# B&R Automation Studio project PLC code - cp (part 9)

#### LocalFunctions.fun
```iecst
{REDUND_ERROR} FUNCTION ModuleStatus : NIRAdphos_ModuleState (*TODO: Add your comment here*) (*$GROUP=User,$CAT=User,$GROUPICON=User.png,$CATICON=User.png*)
	VAR_INPUT
		StatusValue : INT;
	END_VAR
END_FUNCTION
```

#### Alarms.st
```iecst
ACTION Alarms:

	//////////////////////////
	////// RESET ALARMS //////
	IF data.Commands.xReset THEN
		data.Alarms := resetedAlarms;
		data.AlSummary := resetedAlarmsSummary;
	END_IF

	IF NOT data.Status.xCommsOK THEN
		data.Alarms.xCommsError := TRUE;
	END_IF

	IF data.Signals.In.xFault THEN
		data.Alarms.xFault := TRUE;
	END_IF

	IF NOT data.Signals.In.xSafetyOK THEN
		data.Alarms.xSafetyError := TRUE;
	END_IF

	//Module alarms
	xAnyBlockedFan := FALSE;
	xAnyJam := FALSE;
	FOR iIndexModule := 1 TO data.Parameters.iTotalModules DO

		//Temperatures
		IF data.Status.rSurfaceTempModule[iIndexModule] > data.Parameters.rMaxSurfaceTemp THEN
			data.Alarms.xMaxSurfaceTempModule[iIndexModule] := TRUE;
		END_IF
		IF data.Signals.In.xSurfaceTempModuleSensorError[iIndexModule] THEN
			data.Alarms.xSurfaceTempModuleSensorError[iIndexModule] := TRUE;
		END_IF

		IF data.Signals.In.Jam[iIndexModule].xMechCross AND data.Orders.xCheckJam THEN
			data.Alarms.Jam[iIndexModule].xMechCross:=TRUE;
		END_IF

		//Jams. Check anyJam
		IF data.Alarms.Jam[iIndexModule].xMechCross THEN
			xAnyJam := TRUE;
		END_IF

		//Blocked Fans
		FOR iIndexFan := 1 TO 4 DO
			IF data.Signals.In.BlockedFans[iIndexModule].Fan[iIndexFan] THEN
				data.Alarms.BlockedFansModule[iIndexModule].Fan[iIndexFan] := TRUE;
				xAnyBlockedFan := TRUE;
			END_IF
		END_FOR

	END_FOR

	data.Alarms.xAnyJam := xAnyJam;

	IF data.Signals.In.xInletHumiditySensorError THEN
		data.Alarms.xInletHumiditySensorError := TRUE;
	END_IF
	IF data.Signals.In.xInletTempSensorError THEN
		data.Alarms.xInletTempSensorError := TRUE;
	END_IF

	/////////////////////////////////////////////////////////////////
	//  SOUND  SOUND  SOUND  SOUND  SOUND  SOUND  SOUND
	/////////////////////////////////////////////////////////////////

	arFault(xAlarm:= data.Alarms.xFault, xSilence:=data.Commands.xMute);
	arSafety(xAlarm:= data.Alarms.xSafetyError, xSilence:=data.Commands.xMute);
	arSurfaceTemp1(xAlarm:= data.Alarms.xMaxSurfaceTempModule[1], xSilence:=data.Commands.xMute);
	arSurfaceTemp2(xAlarm:= data.Alarms.xMaxSurfaceTempModule[2], xSilence:=data.Commands.xMute);
	arSurfaceTempSensorError1(xAlarm:= data.Alarms.xSurfaceTempModuleSensorError[1], xSilence:=data.Commands.xMute);
	arSurfaceTempSensorError2(xAlarm:= data.Alarms.xSurfaceTempModuleSensorError[2], xSilence:=data.Commands.xMute);
	arAnyBlockedFan(xAlarm:= xAnyBlockedFan, xSilence:=data.Commands.xMute);
	arAnyJam(xAlarm:= xAnyJam, xSilence:=data.Commands.xMute);

	reasonSound.0 := arFault.xAlarmSound;
	reasonSound.1 := arSafety.xAlarmSound;
	reasonSound.2 := arSurfaceTemp1.xAlarmSound;
	reasonSound.3 := arSurfaceTemp2.xAlarmSound;
	reasonSound.4 := arSurfaceTempSensorError1.xAlarmSound;
	reasonSound.5 := arSurfaceTempSensorError2.xAlarmSound;
	reasonSound.6 := arAnyBlockedFan.xAlarmSound;
	reasonSound.7 := arAnyJam.xAlarmSound;

	data.AlSummary.xAlarmSound := reasonSound>0;

END_ACTION
```

#### AlarmsSummary.st
```iecst
ACTION AlarmsSummary:

	iReasonStop.0 := data.Alarms.xCommsError;
	iReasonStop.1 := data.Alarms.xMaxSurfaceTempModule[1];
	iReasonStop.2 := data.Alarms.xMaxSurfaceTempModule[2];
	iReasonStop.3 := data.Alarms.xFault;
	iReasonStop.4 := data.Alarms.xAnyJam;
	iReasonStop.5 := data.Alarms.xOpcUaWriteError[1] AND data.Status.xEnabledDDC;
	iReasonStop.6 := data.Alarms.xOpcUaWriteError[2] AND data.Status.xEnabledDDC;
	iReasonStop.7 := FALSE;

	data.AlSummary.xAlarmStop := iReasonStop > 0 AND data.Status.xEnabledNir;
	IF EDGEPOS(data.AlSummary.xAlarmStop) THEN
		data.AlSummary.iReasonStop[0] := iReasonStop;
		LogStopAlarm;
	ELSIF EDGEPOS(NOT data.Parameters.AutoMode.xStop AND NOT data.AlSummary.xAlarmStop) THEN
		data.AlSummary.iReasonStop[0] := 0;
	END_IF

	iReasonCritical.0 := data.Status.Comms.Modules[1].error;
	iReasonCritical.1 := data.Status.Comms.Modules[2].error;
	iReasonCritical.2 := data.Alarms.xSafetyError;

	data.AlSummary.xAlarmCritical := iReasonCritical > 0 AND data.Status.xEnabledNir;
	IF EDGEPOS(data.AlSummary.xAlarmCritical) THEN
		data.AlSummary.iReasonCritical := iReasonCritical;
		LogCriticalAlarm;
	ELSIF EDGEPOS(data.Parameters.StateMode=PRINTERGEN_AUTO AND NOT data.AlSummary.xAlarmCritical) THEN
		data.AlSummary.iReasonCritical := 0;
	END_IF

	// It is just used for drive alarms
	iAnyAlarm.0 := iReasonStop > 0;
	iAnyAlarm.1 := iReasonCritical > 0;
	data.AlSummary.xAnyAlarm:= 	iAnyAlarm > 0;

	// It is just used for drive alarms
	iAnyWarning.0 := FALSE;
	data.AlSummary.xAnyWarning:= iAnyWarning > 0;

END_ACTION
```

#### Calculations.st
```iecst
ACTION Calculations:

	//Avoid access out of the array
	data.Parameters.iTotalModules := MIN(data.Parameters.iTotalModules, MAX_LAST_NIR_MODULES);
	data.Parameters.DDC.iLampsExtend := MIN(data.Parameters.DDC.iLampsExtend, 3); //Limit to 3 as make no sense allow higher values

	data.Status.Comms.xBeltRunning := data.Status.Comms.Speed > 1;

	//Calculation of Modules data
	FOR iIndexModule := 1 TO data.Parameters.iTotalModules DO
		data.Status.rSurfaceTempModule[iIndexModule] := INT_TO_REAL(data.Signals.In.iSurfaceTempModuleRaw[iIndexModule])/10.0;
		data.Status.Comms.Modules[iIndexModule].xPowered := data.Status.Comms.Modules[iIndexModule].Power > 1;
		data.Status.Comms.Modules[iIndexModule].NirStatus := ModuleStatus(data.Status.Comms.Modules[iIndexModule].iNirStatus);

		//Limitation of wrong data in parameters
		data.Parameters.Comms.Modules[iIndexModule].Adjust := LIMIT(-100, data.Parameters.Comms.Modules[iIndexModule].Adjust, 100);
	END_FOR;

	data.Status.xDrying := data.State = NIRADPEW_RUNNING;

	// -40C to +60C Probe. 100C Range
	data.Status.rInletTemperature := ((INT_TO_REAL(data.Signals.In.iInletTempRaw)* 100.0)/32767.0)-40.0;
	data.Status.rInletHumidity := ((INT_TO_REAL(data.Signals.In.iInletHumidityRaw)* 100.0)/32767.0)-0.0;

	//Limitations of values to remain consistent
	data.Parameters.Comms.Pstart := MAX(data.Parameters.Comms.Pstart, 0);
	data.Parameters.Comms.Pend := MIN(data.Parameters.Comms.Pend, 100);

	data.Parameters.Comms.Pstart := MIN(data.Parameters.Comms.Pend,data.Parameters.Comms.Pstart);
	data.Parameters.Comms.Pend := MAX(data.Parameters.Comms.Pend,data.Parameters.Comms.Pstart);
	data.Parameters.Comms.Vstart := MIN(data.Parameters.Comms.Vend,data.Parameters.Comms.Vstart);
	data.Parameters.Comms.Vend := MAX(data.Parameters.Comms.Vend,data.Parameters.Comms.Vstart);

	IF data.Parameters.rBeltSpeed > data.Parameters.Comms.Vstart THEN
		data.Status.rPowerSetPoint := data.Parameters.Comms.Pstart +
								(data.Parameters.rBeltSpeed-data.Parameters.Comms.Vstart) *
								(data.Parameters.Comms.Pend-data.Parameters.Comms.Pstart) /
								(data.Parameters.Comms.Vend-data.Parameters.Comms.Vstart);

		IF data.Parameters.xLineEmptyingBelt THEN
			data.Status.rPowerSetPoint := data.Status.rPowerSetPoint * 0.5;
		END_IF
	ELSE
		data.Status.rPowerSetPoint := 0;
	END_IF

END_ACTION
```

#### CommsBase.st
```iecst
ACTION CommsNir1base:

	(* UA_Write - call methode *)
	IndexRange_Nir1.StartIndex := 0;
	IndexRange_Nir1.EndIndex := 47;
	NodeAddInfo_Nir1.AttributeId := UAAI_Value;
	NodeAddInfo_Nir1.IndexRangeCount := 1;
	NodeAddInfo_Nir1.IndexRange[0] := IndexRange_Nir1;
	UA_Write_Nir1(Execute := ExecuteMethodCall_Nir1,
		ConnectionHdl := ConnectionHdl_Nir1,
		NodeHdl := NodeHdl_Nir1,
		NodeAddInfo := NodeAddInfo_Nir1,
		Timeout := T#10s,
		Variable := '::NIRAdphosC.iValues_Nir1'
	);
	IF NOT UA_Write_Nir1.Busy THEN
		ExecuteMethodCall_Nir1 := FALSE;
		IF UA_Write_Nir1.Done THEN
			NewMediaData_Nir1.rLength := NewMediaData_Nir1.rLength + 1;
		END_IF
		IF UA_Write_Nir1.Error THEN
			NewMediaData_Nir1.rDocLength := NewMediaData_Nir1.rDocLength + 1;
		END_IF
	END_IF

//	// Managing the automatic sending. Not sending if enable drying. Sendign Energy then
//	IF NOT gThicknessCtrl.status.xNewMediaStackEnabled OR gThicknessCtrl.parameters.Dry.xDryStack THEN
//		RETURN;
//	END_IF
//
//	IF (gSimMachine.Parameters.Stack.iMediaQuantityToKeepLoaded <= gThicknessCtrl.status.Stack.iNewMediaLoadedL1 + gThicknessCtrl.status.Stack.iNewMediaLoadedL2) THEN
//		RETURN;
//	END_IF

	// Adding a timer to avoid not working the method
//	tonNotCallingMethod_Nir1.IN := NOT UA_Write_Nir1.Busy;
//	tonNotCallingMethod_Nir1.PT := t#4500ms;
//	tonNotCallingMethod_Nir1();
//	IF EDGEPOS(tonNotCallingMethod_Nir1.Q) THEN
//		ExecuteMethodCall_Nir1 := TRUE;
//	END_IF

	IF xReConnect THEN
		PreparingMethodCommsNir1base;
	END_IF

END_ACTION

ACTION InitialDataForMediaNir1base:

END_ACTION

ACTION PreparingMethodCommsNir1base:

	ExecuteConnect_Nir1 := TRUE;

	(* UA_Connect - establish connection to OPC UA Server *)
	SessionConnectInfo_Nir1.SecurityMsgMode := UASecurityMsgMode_None;
	SessionConnectInfo_Nir1.SecurityPolicy := UASecurityPolicy_None;
	SessionConnectInfo_Nir1.TransportProfile := UATP_UATcp;
	SessionConnectInfo_Nir1.UserIdentityToken.UserIdentityTokenType := UAUITT_Anonymous;
	//SessionConnectInfo_Nir1.UserIdentityToken.TokenParam1 := 'PressCore';
	//SessionConnectInfo_Nir1.UserIdentityToken.TokenParam2 := 'h98o76';
	SessionConnectInfo_Nir1.SessionTimeout := T#1m;
	SessionConnectInfo_Nir1.MonitorConnection := T#10s;

	UA_Connect_Nir1(Execute := ExecuteConnect_Nir1,
		ServerEndpointUrl := 'opc.tcp://192.168.125.91:4840',
	SessionConnectInfo := SessionConnectInfo_Nir1,
	Timeout := T#10s);
	IF NOT UA_Connect_Nir1.Busy THEN
		ExecuteConnect_Nir1 := FALSE;
		IF UA_Connect_Nir1.Done THEN
			ConnectionHdl_Nir1 := UA_Connect_Nir1.ConnectionHdl;
			////// NEXT
			ExecuteGetnamespaceindex_Nir1 := TRUE;
		END_IF
		IF UA_Connect_Nir1.Error THEN
			ConnectionHdl_Nir1 := 0;
		END_IF
	END_IF

	(* UA_GetNamespaceIndex - read index of required namespace for PVs *)
	UA_GetNamespaceIndex_Nir1(Execute := ExecuteGetnamespaceindex_Nir1,
		ConnectionHdl := ConnectionHdl_Nir1,
		NamespaceUri := 'http://opcfoundation.org/UA/',
		Timeout := T#5s);
	IF NOT UA_GetNamespaceIndex_Nir1.Busy THEN
		ExecuteGetnamespaceindex_Nir1 := FALSE;
		IF UA_GetNamespaceIndex_Nir1.Done THEN
			NamespaceIndex_Nir1 := UA_GetNamespaceIndex_Nir1.NamespaceIndex;
			////// NEXT
			ExecuteMethodGetHandle_Nir1 := TRUE;
		END_IF
		IF UA_GetNamespaceIndex_Nir1.Error THEN
			NamespaceIndex_Nir1 := 0;
		END_IF
	END_IF

	(* UA_NodeGetHandle - get a handle for required methode *)
	ObjectNodeID_Nir1.NamespaceIndex := NamespaceIndex_Nir1;
	IF NodeHdl_Nir1 = 0 THEN
		ObjectNodeID_Nir1.Identifier := '26';
		ObjectNodeID_Nir1.IdentifierType := UAIdentifierType_Numeric;
	END_IF

	//MethodNodeID_Nir1.NamespaceIndex := NamespaceIndex_Nir1;
	//MethodNodeID_Nir1.Identifier := '::ThickPos:LoadNewMedia';
	//MethodNodeID_Nir1.IdentifierType := UAIdentifierType_String;
	UA_NodeGetHandle_Nir1(Execute := ExecuteMethodGetHandle_Nir1,
		ConnectionHdl := ConnectionHdl_Nir1,
		NodeID := ObjectNodeID_Nir1,
		//MethodNodeID := MethodNodeID_Nir1,
		Timeout := T#10s);
	IF NOT UA_NodeGetHandle_Nir1.Busy THEN
		ExecuteMethodGetHandle_Nir1 := FALSE;
		IF UA_NodeGetHandle_Nir1.Done THEN
			NodeHdl_Nir1 := UA_NodeGetHandle_Nir1.NodeHdl;
			xReConnect := FALSE;
			////// NEXT
			// READY TO COMMUNICATE
		END_IF
		IF UA_NodeGetHandle_Nir1.Error THEN
			NodeHdl_Nir1 := 0;
			xReConnect := FALSE;
		END_IF
	END_IF

	iTimes := iTimes + 1;

END_ACTION
```

#### NIRAdphosCtrl.st
```iecst
PROGRAM _INIT
	data ACCESS ADR(gNirAdphos);
	//Activate this signal because it not exist physically
	data.Signals.In.xSafetyOK := TRUE;

	InitialDataForMediaNir1;
	//PreparingMethodCommsNir1;
	data.Parameters.DDC.pIntensityNir1 := 0;
	data.Parameters.DDC.pIntensityNir2 := 0;

END_PROGRAM

PROGRAM _CYCLIC

	data ACCESS ADR(gNirAdphos);

	Calculations;

	//Consider the parametrization to use NIR or not when ready
	IF (data.State = NIRADPEW_NOT_INITIALIZED OR data.State = NIRADPEW_IDLE) THEN
		data.Status.xEnabledNir := data.Parameters.xEnableNir AND data.Status.xAnyModuleEnabled;
		data.Status.xEnabledDDC := data.Parameters.DDC.xEnableDDC AND data.Status.xAnyModuleEnabled;
	END_IF

	State;

	Alarms;

	AlarmsSummary;

	Outputs;

	CommsNir1;
	CommsNir2;

END_PROGRAM
```

#### NirFunctions.st
```iecst
(* Return Enum from INT value from comms
NIRAdphos_ModuleState
 NIRADPM_OFF				0
 NIRADPM_STARTUP			1
 NIRADPM_READY				2
 NIRADPM_STANDBY			3
 NIRADPM_PROCESS			4
 NIRADPM_SHUTDOWN			5

*)
FUNCTION ModuleStatus
	CASE StatusValue OF
		0: ModuleStatus := NIRADPM_OFF;
		1: ModuleStatus := NIRADPM_STARTUP;
		2: ModuleStatus := NIRADPM_READY;
		3: ModuleStatus := NIRADPM_STANDBY;
		4: ModuleStatus := NIRADPM_PROCESS;
		5: ModuleStatus := NIRADPM_SHUTDOWN;
		ELSE ModuleStatus := NIRADPM_UNDEFINED;
	END_CASE
END_FUNCTION
```

### NirAdphosSim.typ
```iecst
TYPE
	NirAdphosSimParameters_typ : 	STRUCT
		CurrentSpeed : REAL; (*Current speed of the Belt in m/min*)
	END_STRUCT;
	NirAdphosSimCommands_typ : 	STRUCT
		CreateError : BOOL;
	END_STRUCT;
	NirAdphosSim_typ : 	STRUCT
		Parameters : NirAdphosSimParameters_typ;
		Commands : NirAdphosSimCommands_typ;
	END_STRUCT;
END_TYPE
```

### Program Logical/ExtPack/_Cure/NIRAdphos/NirAdphosSim/NirAdphosSim_v1/NirAdphosSim (IEC)

#### NirAdphosSim.var - Local variables
```iecst
VAR
	SimNirAdphos : REFERENCE TO NirAdphosSim_typ;
	dataNir : REFERENCE TO NIRAdphos;
	tonPowerOn : TON;
	tonReady : TON;
	tonBeltRunning : TON;
	tonDry : TON;
	StatusCommsReseted : NIRAdphos_CommsIn;
	tonCommand : TON;
	iIndexLamp : USINT;
	iIndexModule : USINT;
	xSimulatingCommand : UINT;
	iSetLampTimes : UINT;
	iReasonBeltRunning : USINT;
	tonDelayTemp : TON;
	iMaxTemperature : INT; (*Value x 10 of Celsius*)
	iMinTemperature : INT; (*Value x 10 of Celsius*)
	rModulePower : ARRAY[0..2] OF REAL;
END_VAR
VAR CONSTANT
	POWER_VARIATION : REAL := 0.2;
END_VAR
VAR
	rModulePowerSetPoint : REAL;
END_VAR
```

### Package Logical/ExtPack/_Cure/ArcLampGEW/ArcLampGew_v1 - Program to control a GEW ArcLamp

### Program Logical/ExtPack/_Cure/ArcLampGEW/ArcLampGew_v1/ArcLampGewCtrl (IEC)

#### AlarmsSummary.st
```iecst
ACTION AlarmsSummary:

	iReasonStop.0 := data.Alarms.xJam;
	iReasonStop.1 := data.Status.Lamps[1].InAlarm;
	iReasonStop.2 := data.Status.Lamps[2].InAlarm;

	data.AlSummary.xAlarmStop := iReasonStop > 0 AND data.Status.xEnabledArcLamp;
	IF EDGEPOS(data.AlSummary.xAlarmStop) THEN
		data.AlSummary.iReasonStop[0] := iReasonStop;
		LogStopAlarm;
	ELSIF EDGEPOS(NOT data.Parameters.AutoMode.xStop AND NOT data.AlSummary.xAlarmStop) THEN
		data.AlSummary.iReasonStop[0] := 0;
	END_IF

	iReasonCritical.0 := data.Alarms.xCommsError;

	data.AlSummary.xAlarmCritical := iReasonCritical > 0 AND data.Status.xEnabledArcLamp;
	IF EDGEPOS(data.AlSummary.xAlarmCritical) THEN
		data.AlSummary.iReasonCritical := iReasonCritical;
		LogCriticalAlarm;
	ELSIF EDGEPOS(data.Parameters.StateMode=PRINTERGEN_AUTO AND NOT data.AlSummary.xAlarmCritical) THEN
		data.AlSummary.iReasonCritical := 0;
	END_IF

	// It is just used for drive alarms
	iAnyAlarm.0 := iReasonStop > 0;
	iAnyAlarm.1 := iReasonCritical > 0;
	data.AlSummary.xAnyAlarm:= 	iAnyAlarm > 0;

	// It is just used for drive alarms
	iAnyWarning.0 := FALSE;
	data.AlSummary.xAnyWarning:= iAnyWarning > 0;

END_ACTION
```

#### ArcLampGew.st
```iecst
PROGRAM _INIT

	IF gDryer.St.HwData.Family = FAMILY_BRAUTOMATIONRUNTIME THEN
		Host := '127.0.0.1';
	ELSE
		Host := '192.168.125.39';
	END_IF

	data ACCESS ADR(gArcLampGew);
	InitialiceCommsObjects;

END_PROGRAM

PROGRAM _CYCLIC

	data ACCESS ADR(gArcLampGew);

	//If ArcLamp is not installed, avoid entering in the code
	IF NOT data.Parameters.xInstalled THEN
		data.Status := resetedStatus;
		data.Signals.Out := resetedOuts;
		data.Alarms := resetedAlarms;
		data.AlSummary := resetedAlarmsSummary;
		RETURN;
	END_IF
	data.Status.xInstalled := TRUE; //It is reseted if it is not installed

	//////////////////////////
	////// RESET ALARMS //////
	IF data.Commands.xReset THEN

		//Send reset to reset alarms by comms if any alarm in selected lamp
		xResetNeeded.0 := data.Status.Lamps[1].InAlarm AND data.Parameters.Lamps[1].Enable;
		xResetNeeded.1 := data.Status.Lamps[2].InAlarm AND data.Parameters.Lamps[2].Enable;
		IF xResetNeeded > 0 THEN
			data.Commands.InternalComms.xResetAll := TRUE;
		END_IF

		data.Alarms := resetedAlarms;
		data.AlSummary := resetedAlarmsSummary;

	END_IF

	IF data.State = ARCLGEW_NOT_INITIALIZED OR data.State = ARCLGEW_IDLE THEN
		data.Status.xEnabledArcLamp := data.Parameters.xEnableArcLamp;
	END_IF
	State;

	Comms;

	Alarms;

	AlarmsSummary;

	Calculations;

	Outputs;

END_PROGRAM

PROGRAM _EXIT
	// Release Client instances
	Client(enable := 0, send := 0);
	ClientPost(enable := 0, send := 0);
END_PROGRAM
```

#### Calculations.st
```iecst
ACTION Calculations:

	FOR iLamp:=1 TO data.Parameters.iLampQuantity DO
		data.Status.Lamps[iLamp].xDrying := data.Status.Lamps[iLamp].LampPowerPercent > 3;
	END_FOR;

	data.Status.xDrying := data.Status.xAnyLampSelected AND data.State = ARCLGEW_RUNNING;
END_ACTION
```

#### Comms.st
```iecst
ACTION Comms:

	//It is here to allow the simulation writing directly over data.Status.CommsStatus and working all properly
	xComsStatusChanged := data.Status.CommsStatus<>commsStatus_copy;
	commsStatus_copy:=data.Status.CommsStatus;

	//Not execute communications if in Simulation and comms disabled
	//In this case, the comms structure will be filled in Simulator
	IF data.Parameters.xDisableComms THEN
		RETURN;
	END_IF;

	//Comms Error definition
	tonErrorComms.IN := commsStatus<>ARCLG_IDLE;
	tonErrorComms.PT := T#4s;
	tonErrorComms();

	tonSendReadSystem.IN := commsStatus=ARCLG_IDLE;
	IF NOT data.Alarms.xCommsError THEN
		tonSendReadSystem.PT := T#2s;
	ELSE
		tonSendReadSystem.PT := T#15s;
	END_IF
	tonSendReadSystem();

	tonDelaySendReadSystem.IN := xReadSystemDelay;
	tonDelaySendReadSystem.PT := t#200ms;
	tonDelaySendReadSystem();

	IF tonSendReadSystem.Q OR tonDelaySendReadSystem.Q THEN
		data.Commands.InternalComms.xReadLampsUv := TRUE;
		xReadSystemDelay := FALSE;
	END_IF

	CASE commsStatus OF

		ARCLG_IDLE:
			IF data.Commands.InternalComms.xReadLamps THEN
				commsStatus:=ARCLG_GET_LAMPS;
				iTimesReadLamps := iTimesReadLamps + 1;
			ELSIF data.Commands.InternalComms.xReadAlerts THEN
				commsStatus:=ARCLG_GET_ALERTS;
				iTimesReadAlerts := iTimesReadAlerts + 1;
			ELSIF data.Commands.InternalComms.xSelectLamp THEN
				commsStatus:=ARCLG_SELEC_LAMP;
				iTimesSelectLamp := iTimesSelectLamp + 1;
			ELSIF data.Commands.InternalComms.xDeSelectLamp THEN
				commsStatus:=ARCLG_DESELEC_LAMP;
				iTimesDeselectLamp := iTimesDeselectLamp + 1;
			ELSIF data.Commands.InternalComms.xStopSelected THEN
				commsStatus:=ARCLG_STOP_SELECTED;
				iTimesStopSelected := iTimesStopSelected + 1;
			ELSIF data.Commands.InternalComms.xStartSelected THEN
				commsStatus:=ARCLG_START_SELECTED;
				iTimesStartSelected := iTimesStartSelected + 1;
			ELSIF data.Commands.InternalComms.xDeselectAll THEN
				commsStatus:=ARCLG_DESELEC_ALL;
				iTimesDeselectAll := iTimesDeselectAll + 1;
			ELSIF data.Commands.InternalComms.xSetPower THEN
				commsStatus:=ARCLG_SET_POWER;
				iTimesSetPower := iTimesSetPower + 1;
			ELSIF data.Commands.InternalComms.xResetAll THEN
				commsStatus:=ARCLG_RESET_ALL;
				iTimesResetAll := iTimesResetAll + 1;
			ELSIF data.Commands.InternalComms.xReadLampsUv THEN
				commsStatus:=ARCLG_GET_LAMPS_UV;
				iTimesReadLampsUv := iTimesReadLampsUv + 1;
			ELSIF data.Commands.InternalComms.xReadSystem THEN
				commsStatus:=ARCLG_GET_SYSTEM;
				iTimesReadSystem := iTimesReadSystem + 1;
			END_IF
			data.Commands.InternalComms := CommsCmdReseted;

		ARCLG_GET_SYSTEM,
		ARCLG_GET_LAMPS,
		ARCLG_GET_LAMPS_UV,
		ARCLG_GET_ALERTS:

			CASE commsSubStatus OF

				ARCLGS_IDLE:
					Responsedata := '';
					LoadRequest;
					commsSubStatus:=ARCLGS_SEND_GET_DATA;

				ARCLGS_SEND_GET_DATA:
					AnalyzeSendGetData;

					// If Comms OK, , comms state is reseted
					// If Comms Error, comms state is reseted when registered

				ARCLGS_PARSE_DATA:

					tonParsingError.IN := JSON_Parse_0.Status = 2;
					tonParsingError.PT := t#500ms;
					tonParsingError();

					JSON_Parse_0();
					IF JSON_Parse_0.Status = 1 THEN
						//Done parsing string.
						LoadReceivedData;
						RegisterGoodComms;

					END_IF

					//Error parsing data.
					IF tonParsingError.Q THEN

						ResetJsonParser;

						lastCommsError.Source := HTTPERROR_PARSINGERROR;
						RegisterErrorComms;

					END_IF

			END_CASE

		ARCLG_RESET_ALL,
		ARCLG_STOP_SELECTED,
		ARCLG_START_SELECTED,
		ARCLG_SELEC_LAMP,
		ARCLG_DESELEC_LAMP,
		ARCLG_DESELEC_ALL,
		ARCLG_SET_POWER:

			CASE commsSubStatus OF

				ARCLGS_IDLE:
					Responsedata := '';
					LoadRequest;
					commsSubStatus:=ARCLGS_SEND_POST_DATA;

				ARCLGS_SEND_POST_DATA:
					IF ClientPost.status = 0 AND ClientPost.httpStatus = HTTPSTATUS_OK AND ClientPost.phase = httpPHASE_RECEIVED THEN
						RegisterGoodComms;
					END_IF

			END_CASE
	END_CASE

	IF tonErrorComms.Q THEN
		//Raise a TimeOut Error
		lastCommsError.Source := HTTPERROR_TIMEOUT;
		RegisterErrorComms;
	END_IF

	//Reassign data when trying to communicate
	IF data.Alarms.xCommsError AND EDGEPOS(commsSubStatus=ARCLGS_SEND_GET_DATA) THEN
		InitialiceCommsObjects;
	END_IF

	Client.send := EDGEPOS(Client.enable);
	Client.enable := commsSubStatus=ARCLGS_SEND_GET_DATA;
	Client();
	IF EDGEPOS(commsSubStatus=ARCLGS_SEND_GET_DATA) THEN iSendClient := iSendClient +1; END_IF

	ClientPost.send := EDGEPOS(ClientPost.enable);
	ClientPost.enable := commsSubStatus=ARCLGS_SEND_POST_DATA;
	ClientPost();
	IF EDGEPOS(commsSubStatus=ARCLGS_SEND_POST_DATA) THEN iSendPost := iSendPost +1; END_IF

	data.Status.CommsStatus := commsStatus;

	sysResp;
	LampsResp;
	UvLampsResp;

	//Store the history of the status to easy the debug
	IF EDGEPOS(data.Alarms.xCommsError) THEN
		FOR iIndexHistory:=iHistoryLines TO 1 BY -1 DO
			ErrorCommsHistory[iIndexHistory]:=ErrorCommsHistory[iIndexHistory-1];
		END_FOR;
		ErrorCommsHistory[0]:= lastCommsError;
	END_IF

END_ACTION

ACTION AnalyzeSendGetData:

	IF Client.status = ERR_FUB_ENABLE_FALSE OR Client.status = ERR_FUB_BUSY OR Client.httpStatus = 0 THEN
		//Waiting the function to finish
		RETURN;
	END_IF

	IF Client.status <> ERR_OK THEN
		//FUB error
		lastCommsError.Source := HTTPERROR_FUNCTION;
		RegisterErrorComms;
		RETURN;
	END_IF

	IF Client.httpStatus <> HTTPSTATUS_OK THEN
		//Get response successful but no response data
		lastCommsError.Source := HTTPERROR_RESPONSE_NODATA;
		RegisterErrorComms;
		RETURN;
	END_IF

	IF Responsedata = '' AND Client.phase = httpPHASE_RECEIVED THEN
		lastCommsError.Source := HTTPERROR_EMPTYDATA;
		RegisterErrorComms;
		RETURN;
	END_IF

	LoadVarInJson;
	ResetJsonParser;
	commsSubStatus:=ARCLGS_PARSE_DATA;

END_ACTION

ACTION RegisterGoodComms:

	ResetCommsStatus;

	data.Alarms.xCommsError := FALSE;
	data.Alarms.Comms := resetedComsAlarms;

END_ACTION

ACTION RegisterErrorComms:

	//Register data just with new errors
	IF NOT data.Alarms.xCommsError THEN
		SaveClientInformation;
	END_IF

	ResetCommsStatus;
	ResetLampsStatus;

	data.Alarms.xCommsError := TRUE;

END_ACTION

ACTION ResetCommsStatus:

	commsStatus:=ARCLG_IDLE;
	commsSubStatus:=ARCLGS_IDLE;

END_ACTION

ACTION ResetLampsStatus:

	FOR iLamp:=1 TO data.Parameters.iLampQuantity DO
		data.Status.Lamps[iLamp].UnitInternalState := 'ErrorComms';
		data.Status.Lamps[iLamp].InAlarm := TRUE;
	END_FOR;

END_ACTION

ACTION SaveClientInformation:

	lastCommsError.HttpStatus := Client.httpStatus;
	lastCommsError.Phase := Client.phase;
	lastCommsError.Response := Responsedata;
	lastCommsError.Status := Client.status;
	lastCommsError.Time := TIME();

	iTimesCommsError := iTimesCommsError + 1;

END_ACTION

ACTION LoadRequest:

	CASE commsStatus OF
		ARCLG_GET_SYSTEM:
			Ressource := 'api/system';
			dataToParse := '{"ArcLampGew:sysRespWrk":';
			memset(ADR(sysRespWrk),0,SIZEOF(sysRespWrk));

		ARCLG_GET_LAMPS:
			Ressource := 'api/lamps/0';
			dataToParse := '{"ArcLampGew:LampsRespWrk":';
			memset(ADR(LampsRespWrk),0,SIZEOF(LampsRespWrk));

		ARCLG_GET_LAMPS_UV:
			Ressource := 'api/lamps/0/uv';
			dataToParse := '{"ArcLampGew:UvLampsRespWrk":';
			memset(ADR(UvLampsRespWrk),0,SIZEOF(UvLampsRespWrk));

		ARCLG_GET_ALERTS:
			Ressource := 'api/lamps/0/alerts';
			dataToParse := '{"ArcLampGew:alertsRespWrk":';
			memset(ADR(alertsRespWrk),0,SIZEOF(alertsRespWrk));

		ARCLG_RESET_ALL:
			Ressource := 'api/lamps/0/reset';
			CleanRequestDataPost;

		ARCLG_STOP_SELECTED:
			Ressource := 'api/lamps/0/stop';
			CleanRequestDataPost;

		ARCLG_START_SELECTED:
			Ressource := 'api/lamps/0/start';
			CleanRequestDataPost;

		ARCLG_SELEC_LAMP:
			//Ressource := 'api/lamps/xx/select';
			Ressource := 'api/lamps/';
			brsitoa(iLampComs, ADR(strAux));
			strcat(ADR(Ressource),ADR(strAux));
			strAux := '/select';
			strcat(ADR(Ressource),ADR(strAux));
			CleanRequestDataPost;

		ARCLG_DESELEC_LAMP:
			//Ressource := 'api/lamps/xx/deselect';
			Ressource := 'api/lamps/';
			brsitoa(iLampComs, ADR(strAux));
			strcat(ADR(Ressource),ADR(strAux));
			strAux := '/deselect';
			strcat(ADR(Ressource),ADR(strAux));
			CleanRequestDataPost;

		ARCLG_DESELEC_ALL:
			Ressource := 'api/lamps/0/deselect';
			CleanRequestDataPost;

		ARCLG_SET_POWER:
			Ressource := 'api/lamps/0/powerramping';

			RequestDataPost := '';
			strAux := '';
			paramURL.enable := TRUE;
			paramURL.pParam := ADR('power');
			brsitoa(data.Parameters.iPowerPerc, ADR(strAux));
			paramURL.pValue := ADR(strAux);
			paramURL.pDest := ADR(RequestDataPost);
			paramURL.destSize := SIZEOF(RequestDataPost);
			paramURL();

			strAux := '';
			paramURL.enable := TRUE;
			paramURL.pParam := ADR('speed');
			brsitoa(100, ADR(strAux));
			paramURL.pValue := ADR(strAux);
			paramURL.pDest := ADR(RequestDataPost);
			paramURL.destSize := SIZEOF(RequestDataPost);
			paramURL();

			ClientPost.requestDataLen := LEN(RequestDataPost);
			brsitoa(LEN(RequestDataPost), ADR(RequestHeaderPost.userLine[5].value));

	END_CASE

END_ACTION

ACTION LoadReceivedData:

	CASE commsStatus OF
		ARCLG_GET_SYSTEM:
			sysResp := sysRespWrk;
		ARCLG_GET_LAMPS:
			LampsResp := LampsRespWrk;
		ARCLG_GET_LAMPS_UV:
			UvLampsResp := UvLampsRespWrk;
			LoadReceivedUvData;
		ARCLG_GET_ALERTS:
			alertsResp := alertsRespWrk;
			LoadStatusWithAlerts;
	END_CASE

END_ACTION

ACTION LoadReceivedUvData:

	iLamp:=1;
	UvLampRespAssigWrk ACCESS ADR(UvLampsResp.Lamp1);
	LoadReceivedUvDataLamp;

	iLamp:=2;
	UvLampRespAssigWrk ACCESS ADR(UvLampsResp.Lamp2);
	LoadReceivedUvDataLamp;

END_ACTION

ACTION LoadReceivedUvDataLamp:

	data.Status.Lamps[iLamp].NodeAddress := UvLampRespAssigWrk.NodeAddress;
	data.Status.Lamps[iLamp].UnitInternalState := UvLampRespAssigWrk.UnitInternalState;
	data.Status.Lamps[iLamp].LampPowerPercent := UvLampRespAssigWrk.LampPowerPercent;
	data.Status.Lamps[iLamp].LampPower := UvLampRespAssigWrk.LampPower;
	data.Status.Lamps[iLamp].PressImpression := UvLampRespAssigWrk.PressImpression;
	data.Status.Lamps[iLamp].PressSpeed := UvLampRespAssigWrk.PressSpeed;
	data.Status.Lamps[iLamp].IsSelected := UvLampRespAssigWrk.IsSelected;
	data.Status.Lamps[iLamp].AlertCount := UvLampRespAssigWrk.AlertCount;
	data.Status.Lamps[iLamp].InAlarm := UvLampRespAssigWrk.AlertCount > 0;
	data.Status.Lamps[iLamp].SensorEmission[1] := UvLampRespAssigWrk.Sensor1Raw;
	data.Status.Lamps[iLamp].SensorEmission[2] := UvLampRespAssigWrk.Sensor2Raw;
	data.Status.Lamps[iLamp].SensorEmission[3] := UvLampRespAssigWrk.Sensor3Raw;
	data.Status.Lamps[iLamp].SensorEmission[4] := UvLampRespAssigWrk.Sensor4Raw;
	data.Status.Lamps[iLamp].SensorEmission[5] := UvLampRespAssigWrk.Sensor5Raw;
	data.Status.Lamps[iLamp].SensorEmission[6] := UvLampRespAssigWrk.Sensor6Raw;
	data.Status.Lamps[iLamp].SensorEmission[7] := UvLampRespAssigWrk.Sensor7Raw;
	data.Status.Lamps[iLamp].SensorEmission[8] := UvLampRespAssigWrk.Sensor8Raw;

END_ACTION

ACTION LoadVarInJson:

	strcat(ADR(dataToParse),ADR(Responsedata));
	strAux := '}';
	strcat(ADR(dataToParse),ADR(strAux));

END_ACTION

ACTION ResetJsonParser:

	//Reset Memory
	memset(ADR(JSON_Parse_0),0,SIZEOF(JSON_Parse_0));
	dataDebug := '';
	dataNotFound := '';

	//Reassign
	JSON_Parse_0.pMessage := ADR(dataToParse);
	JSON_Parse_0.pDebug := ADR(dataDebug);
	JSON_Parse_0.SizeDebug := SIZEOF(dataDebug);
	JSON_Parse_0.pVariablesNotFound := ADR(dataNotFound);
	JSON_Parse_0.SizeVariablesNotFound := SIZEOF(dataNotFound);

END_ACTION

ACTION LoadStatusWithAlerts:

	FOR iLamp:=1 TO data.Parameters.iLampQuantity DO
		IF data.Parameters.Lamps[iLamp].Enable THEN
			xAuxVar := FALSE;
			FOR iAlert:=1 TO MAXIMUM_QUANTITY_ALERTS DO
				//TOREVIEW: Do it in reflection
			END_FOR;
		END_IF
	END_FOR;

END_ACTION

ACTION CleanRequestDataPost:

	RequestDataPost := '';
	ClientPost.requestDataLen := 0;
	brsitoa(0, ADR(RequestHeaderPost.userLine[5].value));

END_ACTION

ACTION InitialiceCommsObjects:

	//Host					:= '192.168.125.39'; //Assigned in the init
	//Ressource 			:= 'api/system'; //Assigned before sending the frame

	Client.method 			:= httpMETHOD_GET;
	Client.option 			:= httpOPTION_HTTP_11;

	Client.pHost 			:= ADR(Host);
	Client.hostPort			:= 9910;
	Client.pUri 			:= ADR(Ressource);
	Client.pResponseData 	:= ADR(Responsedata);
	Client.responseDataSize := SIZEOF(Responsedata);
	Client.pRequestHeader	:= ADR(RequestHeader);

	//credentialsFlat	:='S20143:425520'; //Code of the first machine
	//credentialsFlat	:='S1111:366390'; //Code of the simulator
	brsstrcpy(ADR(credentialsUserInternal),ADR(data.Parameters.SerialNumber));
	strAuxCredentials := ':';
	brsstrcat(ADR(credentialsUserInternal), ADR(strAuxCredentials));
	brsstrcat(ADR(credentialsUserInternal), ADR(data.Parameters.PIN));
	brsstrcpy(ADR(credentialsFlat),ADR(credentialsUserInternal));

	authenticationBase		:='Basic ';

	CredentialsEncoder.enable := TRUE;
	CredentialsEncoder.pSrc := ADR(credentialsFlat);
	CredentialsEncoder.srcLen := LEN(credentialsFlat);
	CredentialsEncoder.pDest := ADR(credentialsBase64);
	CredentialsEncoder.destSize := SIZEOF(credentialsBase64);
	CredentialsEncoder();

	RequestHeader.connection := 'keep-alive';

	RequestHeader.userLine[0].name := 'Authorization';
	RequestHeader.userLine[0].value := authenticationBase;
	strcat(ADR(RequestHeader.userLine[0].value),ADR(credentialsBase64));

	RequestHeader.userLine[1].name := 'Content-Type';
	RequestHeader.userLine[1].value := 'text/json';

	RequestHeader.userLine[2].name := 'Accept-Encoding';
	RequestHeader.userLine[2].value := 'gzip, deflate, br';

	RequestHeader.userLine[3].name := 'Host';
	RequestHeader.userLine[3].value := Host;
	strAux := ':';
	strcat(ADR(RequestHeader.userLine[3].value),ADR(strAux));
	itoa(Client.hostPort, ADR(strAux));
	strcat(ADR(RequestHeader.userLine[3].value),ADR(strAux));

	ClientPost.method 			:= httpMETHOD_POST;
	ClientPost.option 			:= httpOPTION_HTTP_11;

	ClientPost.pHost 			:= ADR(Host);
	ClientPost.hostPort			:= 9910;
	ClientPost.pUri 			:= ADR(Ressource);
	ClientPost.pResponseData 	:= ADR(Responsedata);
	ClientPost.responseDataSize := SIZEOF(Responsedata);
	ClientPost.pRequestHeader	:= ADR(RequestHeaderPost);
	ClientPost.pRequestData		:= ADR(RequestDataPost);

	RequestHeaderPost.connection := 'keep-alive';

	RequestHeaderPost.userLine[0].name := 'Authorization';
	RequestHeaderPost.userLine[0].value := authenticationBase;
	strcat(ADR(RequestHeaderPost.userLine[0].value),ADR(credentialsBase64));

	RequestHeaderPost.userLine[1].name := 'Content-Type';
	RequestHeaderPost.userLine[1].value := 'text/json';

	RequestHeaderPost.userLine[2].name := 'Accept-Encoding';
	RequestHeaderPost.userLine[2].value := 'gzip, deflate, br';

	RequestHeaderPost.userLine[3].name := 'Host';
	RequestHeaderPost.userLine[3].value := Host;
	strAux := ':';
	strcat(ADR(RequestHeaderPost.userLine[3].value),ADR(strAux));
	itoa(Client.hostPort, ADR(strAux));
	strcat(ADR(RequestHeaderPost.userLine[3].value),ADR(strAux));

	RequestHeaderPost.userLine[4].name := 'Accept';
	RequestHeaderPost.userLine[4].value := '*/*';

	RequestHeaderPost.userLine[5].name := 'Content-Length';
	//brsitoa(0, ADR(RequestHeaderPost.userLine[5].value)); //Assigned later

	data.Parameters.Lamps[1].Enable := TRUE;
	data.Parameters.Lamps[2].Enable := TRUE;
	data.Parameters.iLampQuantity := 2;

END_ACTION
```

#### EventLog.st
```iecst
ACTION LogStopAlarm:

//	iReasonStop.0 := FALSE;
//	iReasonStop.1 := data.Status.Lamps[1].InAlarm;
//	iReasonStop.2 := data.Status.Lamps[2].InAlarm;
//	iReasonStop.3 := data.Status.Lamps[3].InAlarm;
//	iReasonStop.4 := data.Status.Lamps[4].InAlarm;
//	iReasonStop.5 := data.Status.Lamps[5].InAlarm;
//	iReasonStop.6 := data.Status.Lamps[6].InAlarm;

	stEventLog.Source := ELOG_TYPE_ARCLAMP;
	stEventLog.Severity:= ELOG_SEVERITY_ERROR;
	stEventLog.Facility:= 0;
	stEventLog.ErrorCode:=0;

	stEventLog.Text := 'ArcLamp.LogStopAlarm';

	IF 		iReasonStop.0 THEN stEventLog.Text := '---';
	ELSIF 	iReasonStop.1 THEN stEventLog.Text := 'Error ArcLamp Lamp1';
	ELSIF 	iReasonStop.2 THEN stEventLog.Text := 'Error ArcLamp Lamp2';
	ELSIF 	iReasonStop.3 THEN stEventLog.Text := 'Error ArcLamp Lamp3';
	ELSIF 	iReasonStop.4 THEN stEventLog.Text := 'Error ArcLamp Lamp4';
	ELSIF 	iReasonStop.5 THEN stEventLog.Text := 'Error ArcLamp Lamp5';
	ELSIF 	iReasonStop.6 THEN stEventLog.Text := 'Error ArcLamp Lamp6';
	END_IF

	gEventLogLoader(EventData := ADR(stEventLog));

END_ACTION

ACTION LogCriticalAlarm:

//	iReasonCritical.0 := data.Alarms.xCommsError;

	stEventLog.Source := ELOG_TYPE_ARCLAMP;
	stEventLog.Severity:= ELOG_SEVERITY_ERROR;
	stEventLog.Facility:= 0;
	stEventLog.ErrorCode:=0;

	stEventLog.Text := 'ArcLamp.LogCriticalAlarm';

	IF 		iReasonCritical.0 THEN stEventLog.Text := 'ArcLamp Error Comms';
	ELSIF 	iReasonCritical.1 THEN stEventLog.Text := '---';
	END_IF

	gEventLogLoader(EventData := ADR(stEventLog));

END_ACTION
```

#### Outputs.st
```iecst
ACTION Outputs:

	data.Signals.Out.xImpression := CurrentState = ARCLGEW_RUNNING AND data.Commands.xMediaInside;

	iReasonToStop.0 := data.Alarms.xJam;
	iReasonToStop.1 := data.Commands.xExternalSafetyStop;
	iReasonToStop.2 := CurrentState = ARCLGEW_RUNNING AND NOT data.Parameters.xBeltRunning;
	data.Signals.Out.xSafetyStop := iReasonToStop=0; //FALSE to Stop

	// 100m/min correspond to 10v
	data.Signals.Out.iBeltSpeed:=REAL_TO_INT(data.Parameters.rBeltSpeed * 32766 / 100.0 ); //10V correspond to 32766units

END_ACTION
```

#### State.st
```iecst
ACTION State:

	xCurrentStateChanged := CurrentState_copy <> CurrentState;
	IF xCurrentStateChanged THEN iStatusChanges := iStatusChanges + 1; END_IF
	CurrentState_copy := CurrentState;

	tonRetryCommand.IN := NOT xCurrentStateChanged AND NOT tonRetryCommand.Q;
	tonRetryCommand.PT := t#400ms;
	tonRetryCommand();

	CASE CurrentState OF
		ARCLGEW_NOT_INITIALIZED:
			IF NOT data.Alarms.xCommsError THEN
				CurrentState := ARCLGEW_INITIALIZING;
			END_IF

		ARCLGEW_COMMS_ERROR:
			IF NOT data.Alarms.xCommsError THEN
				CurrentState := ARCLGEW_INITIALIZING;
			END_IF

		ARCLGEW_INITIALIZING:
			IF NOT data.Status.xAnyLampInError THEN
				CurrentState := ARCLGEW_IDLE;
			END_IF

		ARCLGEW_IDLE:
			IF data.Commands.xPrepare AND data.Status.xAnyLampSelected THEN
				data.Commands.xPrepare := FALSE;
				CurrentState := ARCLGEW_DESELEC;
			END_IF
			data.Commands.xStart := FALSE;
			data.Commands.xStop := FALSE;

		ARCLGEW_DESELEC:
			IF xCurrentStateChanged OR tonRetryCommand.Q THEN
				data.Commands.InternalComms.xDeselectAll := TRUE;
			END_IF

			//After sending a deselec, send a read to read if lamps have beed deselected
			IF data.Status.CommsStatus=ARCLG_IDLE AND commsStatus_copy=ARCLG_DESELEC_ALL THEN
				//data.Commands.InternalComms.xReadLampsUv;
				xReadSystemDelay := TRUE;
			END_IF

			//Go ahead when really deselected
			IF NOT data.Status.Lamps[1].IsSelected AND NOT data.Status.Lamps[2].IsSelected THEN
				CurrentState := ARCLGEW_SELECTING;
			END_IF

		ARCLGEW_SELECTING:
			IF xCurrentStateChanged THEN
				iLampComs:=1;
				PrepareNextEnabledLamp;
			END_IF

			IF tonRetryCommand.Q THEN
				data.Commands.InternalComms.xSelectLamp := TRUE;
			END_IF

			//After a communication, review next steps
			IF data.Status.CommsStatus=ARCLG_IDLE AND commsStatus_copy=ARCLG_SELEC_LAMP THEN
				//If finish communication with the last lamp, ask to review status
				data.Commands.InternalComms.xReadLampsUv := TRUE;

				IF data.Status.Lamps[iLampComs].IsSelected THEN
					IF (iLampComs = iMaxLampSelected) THEN
						CurrentState := ARCLGEW_SET_PARAMS;
					ELSE
						iLampComs := iLampComs + 1;
						PrepareNextEnabledLamp;
					END_IF
				END_IF
			END_IF

		ARCLGEW_SET_PARAMS:
			IF xCurrentStateChanged OR tonRetryCommand.Q THEN
				data.Commands.InternalComms.xSetPower := TRUE;
			END_IF
			IF data.Status.CommsStatus=ARCLG_IDLE AND commsStatus_copy=ARCLG_SET_POWER THEN
				CurrentState := ARCLGEW_SEND_START;
			END_IF

		ARCLGEW_SEND_START:
			IF xCurrentStateChanged OR tonRetryCommand.Q THEN
				data.Commands.InternalComms.xStartSelected := TRUE;
			END_IF
			IF data.Status.CommsStatus=ARCLG_IDLE AND commsStatus_copy=ARCLG_START_SELECTED THEN
				CurrentState := ARCLGEW_STARTING;
			END_IF

		ARCLGEW_STARTING:

			tonInputReady.IN := NOT xCurrentStateChanged AND data.Signals.In.xReady;
			tonInputReady.PT := t#500ms;
			tonInputReady();

			IF data.Commands.xStop THEN
				data.Commands.xStop := FALSE;
				CurrentState := ARCLGEW_SEND_STOP;
			ELSIF tonInputReady.Q THEN
				CurrentState := ARCLGEW_READY;
			END_IF

		ARCLGEW_READY:
			IF data.Commands.xStop THEN
				data.Commands.xStop := FALSE;
				CurrentState := ARCLGEW_SEND_STOP;
			ELSIF data.Commands.xStart THEN
				data.Commands.xStart := FALSE;
				CurrentState := ARCLGEW_RUNNING;
			END_IF

		ARCLGEW_RUNNING:
			IF data.Commands.xStop THEN
				data.Commands.xStop := FALSE;
				CurrentState := ARCLGEW_SEND_STOP;
			END_IF

		ARCLGEW_SEND_STOP:
			IF xCurrentStateChanged OR tonRetryCommand.Q THEN
				data.Commands.InternalComms.xStopSelected := TRUE;
			END_IF

			tonInputReady.IN := NOT xCurrentStateChanged AND NOT data.Signals.In.xReady;
			tonInputReady.PT := t#500ms;
			tonInputReady();

			IF tonInputReady.Q THEN
				CurrentState := ARCLGEW_IDLE;
			END_IF

		ARCLGEW_ERROR:
			IF NOT data.Signals.In.xFault THEN
				CurrentState := ARCLGEW_IDLE;
			END_IF

	END_CASE

	IF data.Alarms.xCommsError THEN
		CurrentState := ARCLGEW_COMMS_ERROR;
	END_IF

	IF data.Signals.In.xFault OR NOT data.Status.xEnabledArcLamp OR data.Parameters.StateMode = PRINTERGEN_ZERO THEN
		CurrentState := ARCLGEW_NOT_INITIALIZED;
	END_IF

	//Store the history of the status to easy the debug
	IF CurrentState<>StateHistory[0] THEN
		FOR iIndexHistory:=iHistoryLines TO 1 BY -1 DO
			StateHistory[iIndexHistory]:=StateHistory[iIndexHistory-1];
		END_FOR;
		StateHistory[0]:=CurrentState;
	END_IF

	data.State := CurrentState;

	//////////////////////////////////////////
	///// AUXILIARY DATA FOR THE TRANSITIONS
	xAnyLampSelected := FALSE;
	iMaxLampSelected := 0;
	FOR iLamp:=1 TO data.Parameters.iLampQuantity DO
		data.Status.Lamps[iLamp].Enabled := data.Parameters.Lamps[iLamp].Enable;
		IF data.Parameters.Lamps[iLamp].Enable THEN
			xAnyLampSelected := TRUE;
			iMaxLampSelected := iLamp;
		END_IF
	END_FOR;
	data.Status.xAnyLampSelected := xAnyLampSelected;

END_ACTION

ACTION PrepareNextEnabledLamp:

	FOR iLamp:=iLampComs TO data.Parameters.iLampQuantity DO
		IF data.Parameters.Lamps[iLamp].Enable THEN
			iLampComs := iLamp;
			EXIT;
		END_IF
	END_FOR;
	data.Commands.InternalComms.xSelectLamp := TRUE;

END_ACTION
```

### WebServices.typ
```iecst
TYPE
	CommsCommands : 	STRUCT
		xReadAlerts : BOOL;
		xReadLamps : BOOL;
		xReadLampsUv : BOOL;
		xReadSystem : BOOL;
		xResetAll : BOOL;
		xSelectLamp : BOOL;
		xDeSelectLamp : BOOL;
		xStopSelected : BOOL;
		xStartSelected : BOOL;
		xDeselectAll : BOOL;
		xSetPower : BOOL;
	END_STRUCT;
	AlertDetailsResp : 	STRUCT
		AlertCode : STRING[80];
		AlertNumber : UDINT;
		IsFault : BOOL;
		IsWarning : BOOL;
	END_STRUCT;
	LampAlertsResp : 	STRUCT
		NodeAddress : UINT;
		Alerts : ARRAY[0..8]OF AlertDetailsResp;
		AlertCount : USINT;
	END_STRUCT;
	AlertsLampResp : 	STRUCT
		Lamp1 : LampAlertsResp;
		Lamp2 : LampAlertsResp;
	END_STRUCT;
	LampResp : 	STRUCT
		NodeAddress : UINT;
		UnitInternalState : STRING[80];
		LampPowerPercent : UINT;
		LampPower : UINT;
		PressImpression : BOOL;
		PressSpeed : UINT;
		IsSelected : BOOL;
		AlertCount : USINT;
	END_STRUCT;
	AllLampsResp : 	STRUCT
		Success : BOOL;
		Lamp1 : LampResp;
		Lamp2 : LampResp;
	END_STRUCT;
	UvLampResp : 	STRUCT
		NodeAddress : UINT;
		UnitInternalState : STRING[80];
		LampPowerPercent : UINT;
		LampPower : UINT; (*Watts*)
		PressImpression : BOOL;
		PressSpeed : UINT; (*%*)
		IsSelected : BOOL;
		AlertCount : USINT;
		Sensor1Raw : USINT; (*100x mW/cm2*)
		Sensor2Raw : USINT; (*100x mW/cm2*)
		Sensor3Raw : USINT; (*100x mW/cm2*)
		Sensor4Raw : USINT; (*100x mW/cm2*)
		Sensor5Raw : USINT; (*100x mW/cm2*)
		Sensor6Raw : USINT; (*100x mW/cm2*)
		Sensor7Raw : USINT; (*100x mW/cm2*)
		Sensor8Raw : USINT; (*100x mW/cm2*)
	END_STRUCT;
	UvStatusResp : 	STRUCT
		Lamp1 : UvLampResp;
		Lamp2 : UvLampResp;
	END_STRUCT;
	SystemResp : 	STRUCT
		RequestURL : STRING[80];
		CurrentDateTime : STRING[80];
		ResponseID : UDINT;
		Success : BOOL;
		ExecutionTime : UDINT;
		SystemSerial : STRING[80];
		SystemDescription : STRING[80];
		CurrentSoftware : STRING[80];
	END_STRUCT;
	HTTP_CLIENT_ERROR_SOURCE :
		(
		HTTPERROR_UNDEFINED,
		HTTPERROR_FUNCTION,
		HTTPERROR_RESPONSE_NODATA,
		HTTPERROR_EMPTYDATA,
		HTTPERROR_TIMEOUT,
		HTTPERROR_PARSINGERROR
		);
	ErrorWebServiceData : 	STRUCT
		Status : UINT;
		HttpStatus : UINT;
		Phase : UINT;
		Response : STRING[6000];
		Source : HTTP_CLIENT_ERROR_SOURCE;
		Time : TIME;
	END_STRUCT;
END_TYPE
```

### ArcLampGew.typ - Local data types
```iecst
TYPE
	ArcLampGew_SubComms :
		(
		ARCLGS_IDLE,
		ARCLGS_SEND_GET_DATA,
		ARCLGS_SEND_POST_DATA,
		ARCLGS_PARSE_DATA
		);
	ArcLampGew_Comms :
		(
		ARCLG_IDLE,
		ARCLG_GET_SYSTEM,
		ARCLG_GET_LAMPS,
		ARCLG_GET_LAMPS_UV,
		ARCLG_GET_ALERTS,
		ARCLG_RESET_ALL,
		ARCLG_STOP_SELECTED,
		ARCLG_START_SELECTED,
		ARCLG_SELEC_LAMP,
		ARCLG_DESELEC_LAMP,
		ARCLG_DESELEC_ALL,
		ARCLG_SET_POWER
		);
	ArcLampGew_State :
		(
		ARCLGEW_NOT_INITIALIZED,
		ARCLGEW_INITIALIZING,
		ARCLGEW_IDLE,
		ARCLGEW_SELECTING,
		ARCLGEW_SET_PARAMS,
		ARCLGEW_SEND_START,
		ARCLGEW_STARTING,
		ARCLGEW_READY,
		ARCLGEW_RUNNING,
		ARCLGEW_SEND_STOP,
		ARCLGEW_DESELEC,
		ARCLGEW_ERROR,
		ARCLGEW_COMMS_ERROR
		);
	ArcLampGew_LampStatus : 	STRUCT
		NodeAddress : UINT;
		UnitInternalState : STRING[80];
		LampPowerPercent : REAL;
		LampPower : REAL; (*Watts*)
		PressImpression : BOOL;
		PressSpeed : UINT; (*%*)
		IsSelected : BOOL;
		AlertCount : USINT;
		xDrying : BOOL;
		InAlarm : BOOL;
		SensorEmission : ARRAY[0..8]OF UINT; (*0 not used. W/cm2*)
		Enabled : BOOL;
	END_STRUCT;
	ArcLampGew_LampParameters : 	STRUCT
		Enable : BOOL;
	END_STRUCT;
	ArcLampGew_Parameters : 	STRUCT
		StateMode : enumEFI_GenMachineState; (*commands to block*)
		AutoMode : stEFI_MachineAutoModes;
		xInstalled : BOOL;
		xEnableArcLamp : BOOL;
		xDisableComms : BOOL; (*Just for Simulation. Comms can be desabled just in Simulation. Always running in machine*)
		CpuFamily : USINT;
		iLampQuantity : USINT; (*Total quantity of lamps installed in the machine*)
		iPowerPerc : USINT; (*Power in Percentage*)
		rBeltSpeed : REAL; (*Current speed of the belt*)
		xBeltRunning : BOOL; (*Belt is running and starting is allowed*)
		Lamps : ARRAY[0..MAX_LAST_GEW_ARCLAMPS]OF ArcLampGew_LampParameters;
		SerialNumber : STRING[80]; (*Serial number of the Rhino*)
		PIN : STRING[80]; (*Pin to communicate with the API*)
	END_STRUCT;
	ArcLampGew_CommsAlarms : 	STRUCT
		xServerError : BOOL;
		xCredentialsError : BOOL;
	END_STRUCT;
	ArcLampGew_Alarms : 	STRUCT
		xCommsError : BOOL;
		xJam : BOOL; (*EFI Sensor*)
		Comms : ArcLampGew_CommsAlarms;
	END_STRUCT;
	ArcLampGew_Commands : 	STRUCT
		xPrepare : BOOL; (*EDGE*)
		xStart : BOOL; (*EDGE*)
		xStop : BOOL; (*EDGE*)
		xMediaInside : BOOL;
		xReset : BOOL;
		xMute : BOOL;
		xExternalSafetyStop : BOOL; (*External Safety Stop order*)
		InternalComms : CommsCommands;
	END_STRUCT;
	ArcLampGew_SignalsIn : 	STRUCT
		xReady : BOOL;
		xFault : BOOL; (*Any error in the enabled alarms*)
		xJam : BOOL; (*EFI sensor*)
	END_STRUCT;
	ArcLampGew_SignalsOut : 	STRUCT
		xImpression : BOOL;
		xSafetyStop : BOOL; (*Any error in the enabled alarms*)
		iBeltSpeed : INT; (*Current speed of the belt*)
	END_STRUCT;
	ArcLampGew_Signals : 	STRUCT
		In : ArcLampGew_SignalsIn;
		Out : ArcLampGew_SignalsOut; (*Any error in the enabled alarms*)
	END_STRUCT;
	ArcLampGew_Status : 	STRUCT
		xInstalled : BOOL; (*The system is or can be installed*)
		xDrying : BOOL; (*Summary information. State == RUNNING*)
		xEnabledArcLamp : BOOL;
		xAnyLampSelected : BOOL;
		xAnyLampInError : BOOL; (*Any error in the enabled alarms*)
		Lamps : ARRAY[0..MAX_LAST_GEW_ARCLAMPS]OF ArcLampGew_LampStatus;
		CommsStatus : ArcLampGew_Comms;
	END_STRUCT;
	ArcLampGew : 	STRUCT
		Parameters : ArcLampGew_Parameters;
		State : ArcLampGew_State := ARCLGEW_NOT_INITIALIZED;
		Alarms : ArcLampGew_Alarms;
		AlSummary : stEFI_AlarmSummary;
		Commands : ArcLampGew_Commands;
		Signals : ArcLampGew_Signals;
		Status : ArcLampGew_Status;
	END_STRUCT;
END_TYPE
```

- ArcLampGewStates.graphml - Photocell states ctrl (not shown)

### Program Logical/ExtPack/_Cure/ArcLampGEW/ArcLampSim/ArcLampSim_v1/ArcLampSim (IEC)

#### ArcLampSim.st
```iecst
PROGRAM _INIT

	dataArcLamp ACCESS ADR(gArcLampGew);

	dataArcLamp.Parameters.iPowerPerc:= 60;

	IF gDryer.St.HwData.Family = FAMILY_BRAUTOMATIONRUNTIME THEN
		dataArcLamp.Parameters.SerialNumber := 'S11111';
		dataArcLamp.Parameters.PIN 			:= '366390';
	END_IF

END_PROGRAM

PROGRAM _CYCLIC
	(* Insert code here *)
	dataArcLamp ACCESS ADR(gArcLampGew);
	SimArcLamp ACCESS ADR(gSimArcLamp);

//	ARCLG_IDLE:
//		IF data.Commands.InternalComms.xReadLamps THEN
//			commsStatus:=ARCLG_GET_LAMPS;
//		ELSIF data.Commands.InternalComms.xReadAlerts THEN
//			commsStatus:=ARCLG_GET_ALERTS;
//		ELSIF data.Commands.InternalComms.xResetAll THEN
//			commsStatus:=ARCLG_RESET_ALL;
//		ELSIF data.Commands.InternalComms.xSelectLamp THEN
//			commsStatus:=ARCLG_SELEC_LAMP;
//		ELSIF data.Commands.InternalComms.xDeSelectLamp THEN
//			commsStatus:=ARCLG_DESELEC_LAMP;
//		ELSIF data.Commands.InternalComms.xStopSelected THEN
//			commsStatus:=ARCLG_STOP_SELECTED;
//		ELSIF data.Commands.InternalComms.xStartSelected THEN
//			commsStatus:=ARCLG_START_SELECTED;
//		ELSIF data.Commands.InternalComms.xDeselectAll THEN
//			commsStatus:=ARCLG_DESELEC_ALL;
//		ELSIF data.Commands.InternalComms.xSetPower THEN
//			commsStatus:=ARCLG_SET_POWER;
//		ELSIF data.Commands.InternalComms.xReadSystem THEN
//			commsStatus:=ARCLG_GET_SYSTEM;
//		END_IF

	FOR iIndexLamp := 1 TO dataArcLamp.Parameters.iLampQuantity DO

		dataArcLamp.Status.Lamps[iIndexLamp].Enabled := dataArcLamp.Parameters.Lamps[iIndexLamp].Enable;
		IF dataArcLamp.State = ARCLGEW_RUNNING THEN
			IF REAL_TO_USINT(dataArcLamp.Status.Lamps[iIndexLamp].LampPowerPercent) < dataArcLamp.Parameters.iPowerPerc THEN
				dataArcLamp.Status.Lamps[iIndexLamp].LampPowerPercent := MIN(dataArcLamp.Status.Lamps[iIndexLamp].LampPowerPercent + 0.5, dataArcLamp.Parameters.iPowerPerc);
			ELSE
				dataArcLamp.Status.Lamps[iIndexLamp].LampPowerPercent := MAX(dataArcLamp.Status.Lamps[iIndexLamp].LampPowerPercent - 0.5, dataArcLamp.Parameters.iPowerPerc);
			END_IF
		ELSE
			dataArcLamp.Status.Lamps[iIndexLamp].LampPowerPercent := MAX(dataArcLamp.Status.Lamps[iIndexLamp].LampPowerPercent - 0.5, 0);
		END_IF
		//dataArcLamp.Status.Lamps[iIndexLamp].xDrying := dataArcLamp.State = ARCLGEW_RUNNING AND dataArcLamp.Status.Lamps[iIndexLamp].Enabled;
	END_FOR;

	IF dataArcLamp.Commands.InternalComms.xDeselectAll THEN
		IF EDGEPOS(dataArcLamp.Commands.InternalComms.xDeselectAll AND dataArcLamp.Status.CommsStatus = ARCLG_IDLE) THEN
			dataArcLamp.Status.CommsStatus := ARCLG_DESELEC_ALL;
			dataArcLamp.Status.Lamps[1].IsSelected := FALSE;
			dataArcLamp.Status.Lamps[2].IsSelected := FALSE;
		END_IF
		EndComms;
	ELSIF dataArcLamp.Commands.InternalComms.xDeSelectLamp THEN
		IF EDGEPOS(dataArcLamp.Commands.InternalComms.xDeSelectLamp AND dataArcLamp.Status.CommsStatus = ARCLG_IDLE) THEN
			dataArcLamp.Status.CommsStatus := ARCLG_DESELEC_LAMP;
			dataArcLamp.Status.Lamps[1].IsSelected := FALSE;
			dataArcLamp.Status.Lamps[2].IsSelected := FALSE;
		END_IF
		EndComms;
	ELSIF dataArcLamp.Commands.InternalComms.xReadAlerts THEN
		IF EDGEPOS(dataArcLamp.Commands.InternalComms.xReadAlerts AND dataArcLamp.Status.CommsStatus = ARCLG_IDLE) THEN
			dataArcLamp.Status.CommsStatus := ARCLG_GET_ALERTS;
		END_IF
		EndComms;
	ELSIF dataArcLamp.Commands.InternalComms.xReadLamps THEN
		IF EDGEPOS(dataArcLamp.Commands.InternalComms.xReadLamps AND dataArcLamp.Status.CommsStatus = ARCLG_IDLE) THEN
			dataArcLamp.Status.CommsStatus := ARCLG_GET_LAMPS;
		END_IF
		EndComms;
	ELSIF dataArcLamp.Commands.InternalComms.xReadSystem THEN
		IF EDGEPOS(dataArcLamp.Commands.InternalComms.xReadSystem AND dataArcLamp.Status.CommsStatus = ARCLG_IDLE) THEN
			dataArcLamp.Status.CommsStatus := ARCLG_GET_SYSTEM;
		END_IF
		EndComms;
	ELSIF dataArcLamp.Commands.InternalComms.xResetAll THEN
		IF EDGEPOS(dataArcLamp.Commands.InternalComms.xResetAll AND dataArcLamp.Status.CommsStatus = ARCLG_IDLE) THEN
			dataArcLamp.Status.CommsStatus := ARCLG_RESET_ALL;
		END_IF
		EndComms;
	ELSIF dataArcLamp.Commands.InternalComms.xSelectLamp THEN
		IF EDGEPOS(dataArcLamp.Commands.InternalComms.xSelectLamp AND dataArcLamp.Status.CommsStatus = ARCLG_IDLE) THEN
			dataArcLamp.Status.CommsStatus := ARCLG_SELEC_LAMP;
			dataArcLamp.Status.Lamps[1].IsSelected := dataArcLamp.Parameters.Lamps[1].Enable;
			dataArcLamp.Status.Lamps[2].IsSelected := dataArcLamp.Parameters.Lamps[2].Enable;
			iSetLampTimes := iSetLampTimes +1;
		END_IF
		EndComms;
	ELSIF dataArcLamp.Commands.InternalComms.xSetPower THEN
		IF EDGEPOS(dataArcLamp.Commands.InternalComms.xSetPower AND dataArcLamp.Status.CommsStatus = ARCLG_IDLE) THEN
			dataArcLamp.Status.CommsStatus := ARCLG_SET_POWER;
		END_IF
		EndComms;
	ELSIF dataArcLamp.Commands.InternalComms.xStartSelected THEN
		IF EDGEPOS(dataArcLamp.Commands.InternalComms.xStartSelected AND dataArcLamp.Status.CommsStatus = ARCLG_IDLE) THEN
			dataArcLamp.Status.CommsStatus := ARCLG_START_SELECTED;
		END_IF
		EndComms;
	ELSIF dataArcLamp.Commands.InternalComms.xStopSelected THEN
		IF EDGEPOS(dataArcLamp.Commands.InternalComms.xStopSelected AND dataArcLamp.Status.CommsStatus = ARCLG_IDLE) THEN
			dataArcLamp.Status.CommsStatus := ARCLG_STOP_SELECTED;
		END_IF
		EndComms;
		IF tonCommand.Q THEN
			dataArcLamp.Signals.In.xReady := FALSE;
		END_IF
	END_IF

	xSimulatingCommand.0 := dataArcLamp.Commands.InternalComms.xDeselectAll ;
	xSimulatingCommand.1 := dataArcLamp.Commands.InternalComms.xDeSelectLamp ;
	xSimulatingCommand.2 := dataArcLamp.Commands.InternalComms.xReadAlerts ;
	xSimulatingCommand.3 := dataArcLamp.Commands.InternalComms.xReadLamps ;
	xSimulatingCommand.4 := dataArcLamp.Commands.InternalComms.xReadSystem ;
	xSimulatingCommand.5 := dataArcLamp.Commands.InternalComms.xResetAll ;
	xSimulatingCommand.6 := dataArcLamp.Commands.InternalComms.xSelectLamp ;
	xSimulatingCommand.7 := dataArcLamp.Commands.InternalComms.xSetPower ;
	xSimulatingCommand.8 := dataArcLamp.Commands.InternalComms.xStartSelected ;
	xSimulatingCommand.9 := dataArcLamp.Commands.InternalComms.xStopSelected ;

	tonCommand.IN := xSimulatingCommand > 0;
	tonCommand.PT := t#300ms;
	tonCommand();

	tonReady.IN := dataArcLamp.State = ARCLGEW_STARTING;
	tonReady.PT:= T#3s;
	tonReady();
	IF tonReady.Q THEN
		dataArcLamp.Signals.In.xReady := TRUE;
	END_IF

//	tonTransport.IN:= dataArcLamp.Outputs.xRunTransport;
//	tonTransport.PT:= T#1s;
//	tonTransport();
//	dataArcLamp.Inputs.xTransportMoving:=tonTransport.Q;
//
//	tonDry.IN:= dataArcLamp.Inputs.xReadyToDry AND dataArcLamp.Outputs.xStartDrying;
//	tonDry.PT:= T#1s;
//	tonDry();
//	dataArcLamp.Inputs.xDrying:=tonDry.Q;
//
//	dataArcLamp.Signals.In.xReady :=TRUE;
//	dataArcLamp.Signals.In.xFault :=FALSE;

END_PROGRAM
```

#### Comms.st
```iecst
ACTION EndComms:

	IF tonCommand.Q	THEN
		dataArcLamp.Status.CommsStatus := ARCLG_IDLE;
		dataArcLamp.Commands.InternalComms := CommsCmdReseted;
	END_IF

END_ACTION
```

### Package Logical/ExtPack/_Transport/BeltCtrl/BeltCtrl_v1 - Belt package

### Program Logical/ExtPack/_Transport/BeltCtrl/BeltCtrl_v1/BeltCtrl (IEC) - Belt program cyclic task

#### BeltManager.var
```iecst
VAR
	iTimesExecutedErrorState : UINT;
	iTimesExecuted : UINT;
END_VAR
VAR CONSTANT
	iHistoryLines : USINT := 20;
END_VAR
VAR
	StateHistory : ARRAY[0..iHistoryLines] OF BeltStates_enum;
	iIndexHistory : USINT;
	iBeltState : BeltStates_enum;
	AxisBelt : REFERENCE TO AxisCtrl_typ; (*Axis control structure*)
	stBeltAlarmSummaryReseted : stEFI_AlarmSummary; (*Reset alarm summary structure*)
	stBeltAlarmsReseted : stBelt_Alarms; (*Reset alarm structure*)
	T_AlrProtDrive : TON;
	ars_AlrStop : AutoResetSound;
	ars_AlrCritical : AutoResetSound;
	ars_AlrWarning : AutoResetSound;
	T_SoundBelt : TON;
	xAnyDriveError : BOOL;
	xRunBeltOrderAfterSound : BOOL; (*Internal to order belt motor after sound*)
	Belt : REFERENCE TO stBelt;
	xRunningState : BOOL;
	iReasonStop : UDINT;
	iReasonCritical : UDINT;
	stEventLogWarning : EventLog_typ;
	stEventLogStop : EventLog_typ;
	stEventLogCritical : EventLog_typ;
END_VAR
VAR RETAIN
	BeltDriveUnit : DriveUnitMngr;
END_VAR
VAR
	tonOvertorqueAlarm : TON;
	TON_OvertorqueWarning : TON;
	iReasonWarning : UINT;
	tonControllerReady : TON;
	iReasonAnyError : USINT;
	tonEnableVoltageSag : TON;
	tpResetAnyDriveAlarm : TP;
	iReasonAutoAcknowledge : UINT;
	xAvoidResettingSafetyErrors : BOOL;
END_VAR
```

#### Alarms.st
```iecst
ACTION Alarms:

	///////////////
	// BELT ALARMS
	///////////////
	// Timer Drive Protection
	T_AlrProtDrive.IN := (NOT Belt.parameters.xDriveProtectionOK);
	T_AlrProtDrive.PT :=T#2s;
	T_AlrProtDrive();
	IF T_AlrProtDrive.Q THEN
		Belt.Al.xAlrProtDrive := TRUE;
	END_IF

	// Alarm: Power Error AND Alarm Drive Protection
	IF AxisBelt.Status.ErrorID=5012 THEN
		Belt.Al.xAlrPowerBeltError := TRUE;
	END_IF

	// Alarm: Comms Error
	IF (AxisBelt.Status.ErrorID=32189) OR (AxisBelt.Status.ErrorID=29265) THEN
		Belt.Al.xAlrComDrive := TRUE;
	END_IF

	//Warning Over Torque
	TON_OvertorqueWarning.IN := ABS(AxisBelt.Status.ActTorque) > AxisBelt.Status.RatedTorque;
	TON_OvertorqueWarning.PT := T#30s;
	TON_OvertorqueWarning();

	IF TON_OvertorqueWarning.Q THEN
		Belt.Al.xWrnOverTorq := TRUE;
	END_IF

	// Alarm: Over Torque
	tonOvertorqueAlarm.IN := ABS(AxisBelt.Status.ActTorque) > AxisBelt.Status.RatedTorque;
	tonOvertorqueAlarm.PT := T#2m;
	tonOvertorqueAlarm();
	IF tonOvertorqueAlarm.Q THEN
		Belt.Al.xAlrOverTorque := TRUE;
	END_IF

	//Alarm: Any error
	iReasonAnyError.0 := AxisBelt.Status.ErrorID<>0 AND (iBeltState<>BELT_NOT_INITIALIZED);
	iReasonAnyError.1 := Belt.Al.xControllerNotReady;
	xAnyDriveError := iReasonAnyError>0;

	Belt.Al.xAnyDriveAlarm := 	xAnyDriveError AND
								NOT Belt.AlSummary.xAlrSafetySystemGeneral AND
								NOT (Belt.commands.Mode.xZero);

	// Alarm: Temp Belt Motor
	Belt.states.rCurrentTemperature := AxisBelt.Status.ActTempMot;
	IF AxisBelt.Status.ActTempMot > (AxisBelt.Status.MaxTempMotor - 5.0) THEN
		IF AxisBelt.Status.MaxTempMotor > 0 THEN Belt.Al.xBeltMotorTemp := TRUE; END_IF
	ELSIF AxisBelt.Status.ActTempMot < (AxisBelt.Status.MaxTempMotor - 7.0) THEN
		Belt.Al.xBeltMotorTemp := FALSE;
	END_IF

	// Alarm: Temp Belt Driver
	IF AxisBelt.Status.ActTempDrv > (AxisBelt.Status.MaxTempDrv - 5.0) THEN
		IF AxisBelt.Status.MaxTempDrv > 0 THEN Belt.Al.xBeltDriverTemp := TRUE; END_IF
	ELSIF AxisBelt.Status.ActTempDrv < (AxisBelt.Status.MaxTempDrv - 7.0) THEN
		Belt.Al.xBeltDriverTemp := FALSE;
	END_IF

	//Alarm: motor parameters from SW
	IF (Belt.parSw.rAxisLength <= 0.0) THEN
		Belt.Al.xAxisLengthNotDefined := TRUE;
	ELSE
		Belt.Al.xAxisLengthNotDefined := FALSE;
	END_IF

	IF (Belt.parSw.rGearBox <= 0.0) THEN
		Belt.Al.xGearBoxNotDefined := TRUE;
	ELSE
		Belt.Al.xGearBoxNotDefined := FALSE;
	END_IF

	tonControllerReady.IN :=	(NOT AxisBelt.Status.ControllerReady OR AxisBelt.Status.ErrorID=29216) AND // ErrorID 29216 3phase input wires disconnected
								NOT Belt.commands.Mode.xZero AND
								NOT Belt.AlSummary.xAlrSafetySystemGeneral;

	tonControllerReady.PT := t#2s;
	tonControllerReady();
	IF tonControllerReady.Q THEN
		Belt.Al.xControllerNotReady := TRUE;
	END_IF

	tonEnableVoltageSag.IN := (AxisBelt.Status.ErrorID=6058 OR AxisBelt.Status.ErrorID=6059) AND NOT Belt.commands.Mode.xZero; // ErrorID 6058 enable1 voltage sag. ErrorID 6059 enable2 voltage sag
	tonEnableVoltageSag.PT := t#300ms;
	tonEnableVoltageSag();
	IF tonEnableVoltageSag.Q THEN
		Belt.Al.xEnableVoltageSag := TRUE;
	END_IF

	//########################## ALARMS SUMMARY ########################################
	AlarmsSummary;
END_ACTION
```

#### EventLog.st
```iecst
ACTION LogStopAlarm:

//	iReasonStop.0 := Belt.Al.xAnyDriveAlarm;
//	iReasonStop.1 := Belt.Al.xAlrComDrive;
//	iReasonStop.2 := Belt.Al.xAlrPowerBeltError;
//	iReasonStop.3 := Belt.Al.xAlrProtDrive;
//	iReasonStop.4 := Belt.Al.xAlrOverTorque;
//	iReasonStop.5 := Belt.Al.xControllerNotReady;
//	iReasonStop.6 := Belt.Al.xEnableVoltageSag;

	stEventLogStop.Source := ELOG_TYPE_BELT;
	stEventLogStop.Severity:= ELOG_SEVERITY_ERROR;
	stEventLogStop.Facility:= 0;
	stEventLogStop.ErrorCode:=0;

	stEventLogStop.Text := 'Belt.LogStopAlarm';

	IF 		iReasonStop.0 THEN stEventLogStop.Text := 'Belt. xAnyDriveAlarm';
	ELSIF 	iReasonStop.1 THEN stEventLogStop.Text := 'Belt. xAlrComDrive';
	ELSIF 	iReasonStop.2 THEN stEventLogStop.Text := 'Belt. xAlrPowerBeltError';
	ELSIF 	iReasonStop.3 THEN stEventLogStop.Text := 'Belt. xAlrProtDrive';
	ELSIF 	iReasonStop.4 THEN stEventLogStop.Text := 'Belt. xAlrOverTorque';
	ELSIF 	iReasonStop.5 THEN stEventLogStop.Text := 'Belt. xControllerNotReady';
	ELSIF 	iReasonStop.6 THEN stEventLogStop.Text := 'Belt. xEnableVoltageSag';
	END_IF

	gEventLogLoader(EventData := ADR(stEventLogStop));

END_ACTION

ACTION LogCriticalAlarm:

//	iReasonCritical.0 := Belt.Al.xAxisLengthNotDefined;
//	iReasonCritical.1 := Belt.Al.xGearBoxNotDefined;

	stEventLogCritical.Source := ELOG_TYPE_BELT;
	stEventLogCritical.Severity:= ELOG_SEVERITY_ERROR;
	stEventLogCritical.Facility:= 0;
	stEventLogCritical.ErrorCode:=0;

	stEventLogCritical.Text := 'Belt.LogCriticalAlarm';

	IF 		iReasonCritical.0 THEN stEventLogCritical.Text := 'Belt. xAxisLengthNotDefined';
	ELSIF 	iReasonCritical.1 THEN stEventLogCritical.Text := 'Belt. xGearBoxNotDefined';
	END_IF

	gEventLogLoader(EventData := ADR(stEventLogCritical));

END_ACTION

ACTION LogWarning:

	stEventLogWarning.Source := ELOG_TYPE_BELT;
	stEventLogWarning.Severity:= ELOG_SEVERITY_INFO;
	stEventLogWarning.Facility:= 0;
	stEventLogWarning.ErrorCode:=0;

	stEventLogWarning.Text := 'Belt.LogWarning';

	IF 	iReasonWarning.0 THEN stEventLogWarning.Text := 'Belt. xBeltMotorTemp';
	ELSIF 	iReasonWarning.1 THEN stEventLogWarning.Text := 'Belt. xBeltDriverTemp';
	ELSIF 	iReasonWarning.2 THEN stEventLogWarning.Text := 'Belt. xWrnOverTorq';
	END_IF

	gEventLogLoader(EventData := ADR(stEventLogWarning));

END_ACTION
```

#### ResetAlarms.st
```iecst
ACTION ResetAlarms:

	Belt.Al:= stBeltAlarmsReseted;
	Belt.AlSummary := stBeltAlarmSummaryReseted;

END_ACTION
```

### Belt.Typ - Belt data type
```iecst
TYPE
	stBelt : 	STRUCT
		commands : stBelt_Commands;
		parameters : stBelt_Parameters;
		parSw : stBelt_SwParameters;
		states : stBelt_States;
		AlSummary : stEFI_AlarmSummary;
		Al : stBelt_Alarms;
		Log : stBelt_Log;
	END_STRUCT;
	stBelt_States : 	STRUCT
		xRuningBelt : BOOL;
		xOrderRuning : BOOL; (*Active when BELT_PREPARING_START OR BELT_RUN_ORDER OR BELT_RUNNING*)
		rCurrentSpeedUnits : REAL; (*Speed in drive units*)
		rCurrentSpeed : REAL; (*Speed in m/min*)
		rMaxTorque : REAL; (*Max Torque of the motor installed to allow sending the Torque as percentage*)
		rTorquePerc : REAL; (*Belt Torque in % over Max torque. gui_q_iCurrentTorque*)
		rCurrentTemperature : REAL; (*Belt temperature in Cº*)
		rMotorPosition : REAL;
		rCurrentTorque : REAL; (*Belt Torque in Newton*meter*)
		rActualCurrent : REAL; (*Current from the Drive in Amps. value Max/Peak*)
		ErrorId : UINT; (*Error in the BeltMotor*)
		State : BeltStates_enum;
		Hw : stBelt_StatusHw;
		rMaxSpeed : REAL; (*Max speed*)
		rMaxTemperature : REAL; (*Motor temp max working temperature*)
		rAcceleration : REAL := 0; (*ramp ACC in mm/s^2 movements. Just working if machine allows it*)
		rDeceleration : REAL := 0; (*ramp DeACC in mm/s^2  movements Just working if machine allows it*)
		MaxNegDeceleration : REAL; (*Rated Torque of the motor in Nm*)
		MaxPosDeceleration : REAL; (*Rated Torque of the motor in Nm*)
		MaxNegAcceleration : REAL; (*Rated Torque of the motor in Nm*)
		MaxPosAcceleration : REAL; (*Rated Torque of the motor in Nm*)
	END_STRUCT;
	stBelt_StatusHw : 	STRUCT
		rMaxSpeed : REAL := 50.0; (*Speed setpoint in m/min*)
	END_STRUCT;
	stBelt_Parameters : 	STRUCT
		IndexAxis : USINT; (*The index of the axis corresponding to the Belt Axis in the machine*)
		DriveUnit : MC_DriveUnitManager;
		xExistBelt : BOOL;
		Direction : USINT; (*direction for commanded movements. 0=Positive 1=Negative*)
		rMaxSpeed : REAL; (*Max speed in m/min depending on the configuration of the machine*)
		rSetPointSpeed : REAL := 20.0; (*Speed setpoint in m/min*)
		xRemoteAcceleration : BOOL; (*Acceleration is configured by Sw*)
		rAcceleration : REAL := 0; (*ramp ACC in mm/s^2 movements*)
		xRemoteDeceleration : BOOL; (*Deceleration is configured by Sw*)
		rSoftDeceleration : REAL := 0; (*ramp DeACC in mm/s^2  movements*)
		rDeceleration : REAL := 0; (*ramp DeACC in mm/s^2  movements*)
		xDriveProtectionOK : BOOL;
		tiTimeBeepBeforeMove : TIME; (*Time beeping before starting the movement*)
		rMaxAcceleration : REAL; (*Max acceleration*)
		rMaxDeceleration : REAL; (*Max deceleration*)
		rMaxGearBox : REAL := 50; (*Max gearbox*)
		rMaxAxisLength : REAL := 1000; (*Max axis length*)
	END_STRUCT;
	stBelt_SwParameters : 	STRUCT
		rAxisLength : REAL := 605.0; (*Roll diameter in mm*)
		rGearBox : REAL := 35.0; (*Reductor received from gui (x:1)*)
		rAcceleration : REAL := 0; (*ramp ACC in mm/s^2 movements. Just working if machine allows it*)
		rDeceleration : REAL := 0; (*ramp DeACC in mm/s^2  movements Just working if machine allows it*)
	END_STRUCT;
	stBelt_Alarms : 	STRUCT
		xAnyDriveAlarm : BOOL; (*ErrorID is different to 0 is generic drive alarm*)
		xAlrPowerBeltError : BOOL; (*gAxisBelt.Status.ErrorID=5012*)
		xAlrComDrive : BOOL; (*gAxisBelt.Status.ErrorID=32189 OR gAxisBelt.Status.ErrorID=29265*)
		xAlrProtDrive : BOOL;
		xAlrOverTorque : BOOL;
		xBeltMotorTemp : BOOL; (*Warning: Belt Motor Temperature Too Hot*)
		xBeltDriverTemp : BOOL; (*Warning: Belt Driver Temperature Too Hot*)
		xWrnOverTorq : BOOL; (*Warning: Belt Over Torque*)
		xAxisLengthNotDefined : BOOL; (*Critical: Motor transmission data not defined*)
		xGearBoxNotDefined : BOOL; (*Critical: Motor transmission data not defined*)
		xControllerNotReady : BOOL; (*Critical: Controller of the Drive not Ready. Usually motor not connected to drive*)
		xEnableVoltageSag : BOOL; (*Critical: Drive enables disabled*)
	END_STRUCT;
	stBelt_Log : 	STRUCT
		iNumberStartStop : BOOL;
		udiKmBand : UDINT;
		iHoursRunning : BOOL;
		diBentTilesBL2 : DINT;
		diBentTilesBL1 : DINT;
	END_STRUCT;
	stBelt_Commands : 	STRUCT
		xRunBelt : BOOL; (*command xRunBelt*)
		xJogBelt : BOOL; (*command xJogBelt. Movement direct without sound*)
		xUseSoftDeceleration : BOOL; (*Command to apply a lower value of deceleration for cases where stop is not critical*)
		xUseJogAccDecc : BOOL; (*Use Jog acceleration and deceleration parameters*)
		xConsentBelt : BOOL; (*Belt Consent state*)
		xExternalSafetyStop : BOOL; (*External Safety Stop order*)
		Mode : StGeneral_States_Mode;
		AutoMode : stEFI_MachineAutoModes; (*commands to inform belt*)
		xMute : BOOL; (*command xMute *)
		xReset : BOOL; (*command xReset*)
	END_STRUCT;
	BeltStates_enum :
		(
		BELT_NOT_INITIALIZED,
		BELT_SWITCH_ON,
		BELT_HOMING,
		BELT_INITIALIZED,
		BELT_IDLE,
		BELT_PREPARING_START,
		BELT_RUN_ORDER,
		BELT_RUNNING,
		BELT_NOT_CONSENT, (*xConsentPrinting,xConsentBypass,xConsentLaboratory and xConsentLine*)
		BELT_ERROR, (*Belt on error*)
		BELT_JOGGING (*Belt been jogged (remotely). No sound. Direct movement*)
		);
END_TYPE
```

### BeltPublicConstants.var - Public constants
```iecst
VAR CONSTANT
	MIN_DURATION_CLEANING_BELT : TIME := T#10S; (*Min time for clean belt duration*)
	MIN_TIME_FOR_CLEANING_TOP_BELT : TIME := T#1M; (*Min time for belt cleaning*)
	MIN_TIME_FOR_CLEANING_BELT : TIME := T#1M; (*Min time for belt cleaning*)
	MIN_TILES_FOR_CLEANING_BELT : UINT := 1; (*min nr tile for clean belt*)
	MIN_DURATION_CLEANING_BELT_TOP : TIME := T#10S; (*Min time for clean belt duration*)
	MIN_TIME_FOR_CLEANING_BELT_TOP : TIME := T#1M; (*Min time for belt cleaning*)
	MIN_TILES_FOR_CLEANING_BELT_TOP : UINT := 1; (*min nr tile for clean belt*)
END_VAR
```

### Belt Docu.txt - Belt package documentation
```
#################################################################################
#################################################################################
#																				#
#			GENERAL USE OF BELT										     		#
#																				#
# 	To use this BELT MANAGER unit, some general variables are needed:			#
#################################################################################

	///////////////////////////
	// Manual movements test
	///////////////////////////

	///////////////////////////
	// Clean belt test
	///////////////////////////
	// INPUTS
	//
	//
	//
	//
	//
	// OUTPUTS
	//
	//
	//
#################################################################################
#################################################################################
#																				#
#			¡¡¡IMPORTANT!!!!													#
# 	Review BELT MANAGER															#
# 																				#
#																				#
#################################################################################
```

- BeltStates.graphml - Belt states graph (not shown)

### Program Logical/ExtPack/_Transport/NonCrashCtrl/NonCrashCtrl_v1/NonCrashCtrl (IEC)

#### StateManager.st
```iecst
ACTION StateManager:

		// ####################################################################
	// ####################################################################
	//
	// Check dataNCStates.graphml to understand better this implementation

	// Here will be implemented a belt states controller,
	CASE StatusCtrl OF

		NONCRASH_NOT_INITIALIZED:
			// PowerOn Command
			IF AxisMotor.Status.ControllerReady THEN
				// Switched on
				AxisMotor.Command.Power:=TRUE;
				StatusCtrl:=NONCRASH_SWITCH_ON;
				AxisMotor.Command.ErrorAcknowledge:= TRUE;
			END_IF

		NONCRASH_SWITCH_ON:

			IF (NOT AxisMotor.Status.HomeOK) AND AxisMotor.Status.PowerOn THEN
				//Doing Home Direct
				StatusCtrl:=NONCRASH_HOMING;
				AxisMotor.Command.HomeDirect :=TRUE;
			ELSIF AxisMotor.Status.HomeOK THEN
				// All is initialized
				StatusCtrl:=NONCRASH_INITIALIZED;
			END_IF;

		NONCRASH_HOMING:
			//Done Home Direct
			IF AxisMotor.Status.HomeOK THEN
				StatusCtrl:=NONCRASH_INITIALIZED;
			END_IF

		NONCRASH_INITIALIZED:
			// dataNC is initialized when axis state is StandStill
			// Waiting for enabled to run state
			IF AxisMotor.Status.PLCopenState.StandStill THEN
				// Ready for movements
				StatusCtrl:=NONCRASH_IDLE;
			ELSIF AxisMotor.Status.PLCopenState.ErrorStop OR AxisMotor.Status.PLCopenState.Disabled THEN
				// Some was wrong!!!
				StatusCtrl:=NONCRASH_ERROR;
			END_IF

		NONCRASH_IDLE:
			// Waiting for movements
			// Command start belt movement
			IF dataNC.Commands.xRun THEN
				StatusCtrl:=NONCRASH_RUN_ORDER;
			END_IF

		NONCRASH_RUN_ORDER:
			//Launched movement
			IF NOT dataNC.Commands.xRun THEN
				StatusCtrl:=NONCRASH_IDLE;

			ELSIF AxisMotor.Status.PLCopenState.ContinuousMotion THEN
				// Waiting for movements
				StatusCtrl:=NONCRASH_RUNNING;
			END_IF

		NONCRASH_RUNNING:
			IF NOT dataNC.Commands.xRun THEN
				StatusCtrl:=NONCRASH_IDLE;
			END_IF

		NONCRASH_ERROR:

			iTimesExecutedErrorState:=iTimesExecutedErrorState+1;

			// Power off
			AxisMotor.Command.Power:=FALSE;

			// Manual recovery:
			AxisMotor.Command.Reset:= dataNC.Commands.xReset AND NOT AxisMotor.Status.ControllerReady;

			//TOREVIEW: Why just acknowledge "known" errors????
			//TOREMOVE: AxisMotor.Command.ErrorAcknowledge:=(AxisMotor.Status.ErrorID = 29209) OR (AxisMotor.Status.ErrorID = 29207);

//			regErrors.0 := AxisMotor.Status.ErrorID = 73;
//			regErrors.1 := AxisMotor.Status.ErrorID = 4005;
//			regErrors.2 := AxisMotor.Status.ErrorID = 5005;
//			regErrors.3 := AxisMotor.Status.ErrorID = 6021;
//			regErrors.4 := AxisMotor.Status.ErrorID = 6023;
//			regErrors.5 := AxisMotor.Status.ErrorID = 6038;
//			regErrors.6 := AxisMotor.Status.ErrorID = 7100;
//			regErrors.7 := AxisMotor.Status.ErrorID = 7215;
//			regErrors.8 := AxisMotor.Status.ErrorID = 29203;
//			regErrors.9 := AxisMotor.Status.ErrorID = 29205;
//			regErrors.10 := AxisMotor.Status.ErrorID = 29206;
//			regErrors.11 := AxisMotor.Status.ErrorID = 29207;
//			regErrors.12 := AxisMotor.Status.ErrorID = 29209;
//			regErrors.13 := AxisMotor.Status.ErrorID = 29216;
//			regErrors.14 := AxisMotor.Status.ErrorID = 29217;
//			regErrors.15 := AxisMotor.Status.ErrorID = 29238;
//			regErrors.16 := AxisMotor.Status.ErrorID = 29226;
//			regErrors.17 := AxisMotor.Status.ErrorID = 32144;
//			regErrors.18 := AxisMotor.Status.ErrorID = 50000;

			AxisMotor.Command.ErrorAcknowledge:= dataNC.Commands.xReset AND AxisMotor.Status.ErrorID<>0;

			IF AxisMotor.Status.ErrorID = 0  THEN
				StatusCtrl:= NONCRASH_NOT_INITIALIZED;
			END_IF

	END_CASE

	/////////////////////////////////
	// Update belt states
	/////////////////////////////////

	// xZero state changes dataNC state to not initialized
	// It avoids transport belt errors
	IF (dataNC.Parameters.Mode.xZero OR NOT dataNC.parSw.xEnable) THEN
		StatusCtrl:=NONCRASH_NOT_INITIALIZED;
		// Error state changes dataNC state
	ELSIF AxisMotor.Status.ErrorID <> 0 OR dataNC.Alarms.xControllerNotReady THEN
		StatusCtrl:=NONCRASH_ERROR;
	END_IF

	dataNC.Status.State := StatusCtrl;

END_ACTION
```

#### Alarms.st
```iecst
ACTION Alarms:

	//Reset Alarms with an external order to reset
	IF dataNC.Commands.xReset THEN
		ResetAlarms;
	END_IF

	//Comms error
	IF (AxisMotor.Status.ErrorID=32189) OR (AxisMotor.Status.ErrorID=29265) THEN
		dataNC.Alarms.xAlrComsDrive := TRUE;
	END_IF

	//If error and not Comms error, defined as Drive Error
	tonAlarmDelay.IN :=  NOT dataNC.Alarms.xAlrComsDrive AND AxisMotor.Status.ErrorID<>0 AND StatusCtrl <> NONCRASH_NOT_INITIALIZED AND NOT dataNC.AlSummary.xAlrSafetySystemGeneral;
	tonAlarmDelay.PT := T#100ms;
	tonAlarmDelay();
	IF tonAlarmDelay.Q THEN
		dataNC.Alarms.xAlrDriveError := TRUE;
	END_IF

	tonOvertorque.IN := AxisMotor.Status.ActTorque > AxisMotor.Status.RatedTorque;
	tonOvertorque.PT := dataNC.Parameters.tiTorqueFilter;
	tonOvertorque();
	IF tonOvertorque.Q THEN
		dataNC.Alarms.xAlrOvertorque := TRUE;
	END_IF

	//Diferential Breaker Alarm
	IF NOT dataNC.Inputs.xDiffContacOk THEN
		dataNC.Alarms.xAlrDiffContact := TRUE;
	END_IF

	//Alarm: motor parameters from SW
	IF (dataNC.parSw.rPerimeter <= 0.0) THEN
		dataNC.Alarms.xPerimeterNotDefined := TRUE;
	ELSE
		dataNC.Alarms.xPerimeterNotDefined := FALSE;
	END_IF

	IF (dataNC.parSw.rGearBox <= 0.0) THEN
		dataNC.Alarms.xGearBoxNotDefined := TRUE;
	ELSE
		dataNC.Alarms.xGearBoxNotDefined := FALSE;
	END_IF

	tonControllerReady.IN := (NOT AxisMotor.Status.ControllerReady OR AxisMotor.Status.ErrorID=29216) AND NOT dataNC.Parameters.Mode.xZero;	//ErrorID 29216 to desconect only power wires
	tonControllerReady.PT := t#300ms;
	tonControllerReady();
	IF tonControllerReady.Q THEN
		dataNC.Alarms.xControllerNotReady := TRUE;
	END_IF

	// SUMMARY SUMMARY SUMMARY SUMMARY SUMMARY SUMMARY SUMMARY SUMMARY
	// SUMMARY SUMMARY SUMMARY SUMMARY SUMMARY SUMMARY SUMMARY SUMMARY

	iReasonStop.0 := dataNC.Alarms.xAlrComsDrive;
	iReasonStop.1 := dataNC.Alarms.xAlrDriveError;
	iReasonStop.2 := dataNC.Alarms.xAlrOvertorque;
	iReasonStop.3 := dataNC.Alarms.xAlrDiffContact;
	iReasonStop.4 := dataNC.Alarms.xControllerNotReady;
	iReasonStop.5 := dataNC.Alarms.xPerimeterNotDefined;
	iReasonStop.6 := dataNC.Alarms.xGearBoxNotDefined;

	dataNC.AlSummary.xAlarmStop:=	iReasonStop > 0;
	IF EDGEPOS(dataNC.AlSummary.xAlarmStop) THEN
		dataNC.AlSummary.iReasonStop[0] := iReasonStop;
		LogStopAlarm;
	ELSIF EDGEPOS(NOT dataNC.Parameters.AutoMode.xStop AND NOT dataNC.AlSummary.xAlarmStop) THEN
		dataNC.AlSummary.iReasonStop[0] := 0;
	END_IF

	dataNC.AlSummary.xAlarmCritical := iReasonCritical > 0;
	IF EDGEPOS(dataNC.AlSummary.xAlarmCritical) THEN
		dataNC.AlSummary.iReasonCritical := iReasonCritical;
	ELSIF EDGEPOS(dataNC.Parameters.Mode.xAuto AND NOT dataNC.AlSummary.xAlarmCritical) THEN
		dataNC.AlSummary.iReasonCritical := 0;
	END_IF

	dataNC.AlSummary.xAlrSafetySystemGeneral := dataNC.Commands.xExternalSafetyStop;

	// SOUND SOUND SOUND SOUND SOUND SOUND SOUND SOUND SOUND SOUND
	// SOUND SOUND SOUND SOUND SOUND SOUND SOUND SOUND SOUND SOUND

	// Reseteable alarms
	arxAlrComsDrive.xAlarm		:= dataNC.Alarms.xAlrComsDrive;
	arxAlrComsDrive.xSilence	:= dataNC.Commands.xMute;
	arxAlrComsDrive();

	arxAlrDriveError.xAlarm		:= dataNC.Alarms.xAlrDriveError;
	arxAlrDriveError.xSilence	:= dataNC.Commands.xMute;
	arxAlrDriveError();

	arxAlrOvertorque.xAlarm		:= dataNC.Alarms.xAlrOvertorque;
	arxAlrOvertorque.xSilence	:= dataNC.Commands.xMute;
	arxAlrOvertorque();

	arxAlrDiffContact.xAlarm	:= dataNC.Alarms.xAlrDiffContact;
	arxAlrDiffContact.xSilence	:= dataNC.Commands.xMute;
	arxAlrDiffContact();

	arxAlrControllerNotReady.xAlarm	:= dataNC.Alarms.xControllerNotReady;
	arxAlrControllerNotReady.xSilence	:= dataNC.Commands.xMute;
	arxAlrControllerNotReady();

	arxAlrPerimeterNotDefined.xAlarm	:= dataNC.Alarms.xPerimeterNotDefined;
	arxAlrPerimeterNotDefined.xSilence	:= dataNC.Commands.xMute;
	arxAlrPerimeterNotDefined();

	arxAlrGearBoxNotDefined.xAlarm	:= dataNC.Alarms.xGearBoxNotDefined;
	arxAlrGearBoxNotDefined.xSilence	:= dataNC.Commands.xMute;
	arxAlrGearBoxNotDefined();

	iReasonSound.0 := arxAlrComsDrive.xAlarmSound;
	iReasonSound.1 := arxAlrDriveError.xAlarmSound;
	iReasonSound.2 := arxAlrOvertorque.xAlarmSound;
	iReasonSound.3 := arxAlrDiffContact.xAlarmSound;
	iReasonSound.4 := arxAlrControllerNotReady.xAlarmSound;
	iReasonSound.5 := arxAlrPerimeterNotDefined.xAlarmSound;
	iReasonSound.6 := arxAlrGearBoxNotDefined.xAlarmSound;
	dataNC.AlSummary.xAlarmSound := iReasonSound > 0;

	// Mute sound in belt alarms
	IF dataNC.Commands.xMute OR dataNC.Commands.xReset THEN
		dataNC.AlSummary.xAlarmSound:= FALSE;
	END_IF

END_ACTION

ACTION ResetAlarms:
	dataNC.Alarms := AlarmsReseted;
	dataNC.AlSummary := AlarmsSummaryReseted;
END_ACTION
```

#### NonCrashCtrl.var - Local variables
```iecst
VAR
	dataNC : REFERENCE TO NonCrash_typ;
	AlarmsSummaryReseted : stEFI_AlarmSummary;
	AlarmsReseted : NonCrashAlarms_typ;
	AxisMotor : REFERENCE TO AxisCtrl_typ;
	StatusCtrl : NonCrashStatusCtrl := NONCRASH_NOT_INITIALIZED;
	iReasonStop : UDINT;
	iReasonCritical : UDINT;
	arxAlrComsDrive : AutoResetSound;
	arxAlrDriveError : AutoResetSound;
	arxAlrOvertorque : AutoResetSound;
	stEventLog : EventLog_typ;
	regErrors : UDINT; (*Registered errors to consider*)
	iTimesExecutedErrorState : UINT;
	DriveUnitManager : DriveUnitMngr;
	xRunningState : BOOL;
	tonOvertorque : TON;
	arxAlrDiffContact : AutoResetSound;
	tonAlarmDelay : TON;
	tonControllerReady : TON;
	arxAlrControllerNotReady : AutoResetSound;
	arxAlrPerimeterNotDefined : AutoResetSound;
	arxAlrGearBoxNotDefined : AutoResetSound;
	iReasonSound : USINT;
END_VAR
```

### Program Logical/ExtPack/_Transport/NonCrashCtrl/NonCrashCtrl_v1/InitNonCrashCtrl (IEC)

#### InitNonCrashCtrl.st - Cyclic code
```iecst
PROGRAM _CYCLIC
	//Init the index to work with
	 iIndexNonCrash := 1;
END_PROGRAM
```

### NonCrash.typ - Local data types
```iecst
TYPE
	NonCrashStatusCtrl :
		(
		NONCRASH_NOT_INITIALIZED,
		NONCRASH_SWITCH_ON,
		NONCRASH_HOMING,
		NONCRASH_INITIALIZED,
		NONCRASH_IDLE,
		NONCRASH_RUN_ORDER,
		NONCRASH_RUNNING,
		NONCRASH_ERROR (*dataNC on error*)
		);
	NonCrashCommands_typ : 	STRUCT
		xRun : BOOL; (*Signal to RUN. Signal to be keep while the running is wanted*)
		xExternalSafetyStop : BOOL; (*External Safety Stop order*)
		xMute : BOOL; (*command xMute *)
		xReset : BOOL; (*command xReset*)
	END_STRUCT;
	NonCrashParametersSw_typ : 	STRUCT
		rSpeedOffset : REAL := 0; (*In m/min. Modification of the speed desired. Fine adjust in commissioning in m/min. gui_i_iNonCrashSpeedOffset*)
		rGearBox : REAL := 0; (*GearBox of the NonCrash axis to allow proper speed calculation*)
		rPerimeter : REAL := 0; (*Perimeter of the NonCrash axis to allow proper speed calculation*)
		xEnable : BOOL; (*Enable the NonCrash in the machines where it can be installed*)
	END_STRUCT;
	NonCrashParameters_typ : 	STRUCT
		xInstalled : BOOL;
		iIndexMotor : USINT; (*Index of the motor in the gAxis[] array*)
		DriveUnit : MC_DriveUnitManager;
		Mode : StGeneral_States_Mode;
		AutoMode : stEFI_MachineAutoModes;
		MotorDirection : MotorDirection_enum; (*To indicate if the motor must spin in reverse*)
		rSpeedSetPoint : REAL := 50.0; (*In m/min Speed SetPoint of the Transport. *)
		rAcceleration : REAL; (*ramp ACC in mm/s^2 movements*)
		rDeceleration : REAL; (*ramp DeACC in mm/s^2  movements*)
		tiTorqueFilter : TIME; (*Time to define the Overtorque if the torque value is higher that the nominal*)
	END_STRUCT;
	NonCrashAlarms_typ : 	STRUCT
		xAlrComsDrive : BOOL; (*Not communication with the Drive of the motor*)
		xAlrDriveError : BOOL; (*Error in the Drive managing the motor*)
		xWrnOvertorque : BOOL; (*Warning. Overtorque in the motor*)
		xAlrOvertorque : BOOL; (*Alarm. Overtorque in the motor*)
		xAlrDiffContact : BOOL; (*Alarm. Diferential contact dripped*)
		xPerimeterNotDefined : BOOL; (*Critical: Motor transmission data not defined*)
		xGearBoxNotDefined : BOOL; (*Critical: Motor transmission data not defined*)
		xControllerNotReady : BOOL; (*Critical: Controller of the Drive not Ready. Usually motor not connected to drive*)
	END_STRUCT;
	NonCrashStatusMotor_typ : 	STRUCT
		xRunning : BOOL; (*The motor is running*)
		rTorque : REAL := 1.0; (*Current torque N·m*)
		rCurrentSpeedUnits : REAL; (*Speed in drive units*)
		rCurrentSpeed : REAL; (*Speed in m/min*)
		ErrorId : UINT; (*Error in the Motor*)
	END_STRUCT;
	NonCrashStatus_typ : 	STRUCT
		State : NonCrashStatusCtrl; (*State of the control*)
		Motor : NonCrashStatusMotor_typ;
		xInstalled : BOOL; (*The system is or can be installed*)
		xEnabled : BOOL; (*The NonCrash in enabled and raises alarms*)
	END_STRUCT;
	NonCrashInputs_typ : 	STRUCT
		xDiffContacOk : BOOL;
	END_STRUCT;
	NonCrash_typ : 	STRUCT
		Commands : NonCrashCommands_typ;
		Parameters : NonCrashParameters_typ;
		parSw : NonCrashParametersSw_typ;
		Status : NonCrashStatus_typ;
		Alarms : NonCrashAlarms_typ; (*Alarms*)
		AlSummary : stEFI_AlarmSummary; (*Alarms Summary*)
		Inputs : NonCrashInputs_typ;
	END_STRUCT;
END_TYPE
```

### NonCrash.var - Local variables
```iecst
VAR
	iIndexNonCrash : USINT;
END_VAR
```

### Program Logical/ExtPack/_Transport/NonCrashCtrl/NonCrashSim/NonCrashSim_v1/InitNonCrashSim (IEC)

#### Cyclic.st
```iecst
PROGRAM _CYCLIC
	(* Insert code here *)
	iNonCrashSimIndex := 1;

END_PROGRAM
```

### NonCrashSim.typ - Local data types
```iecst
TYPE
	SimNonCrashCommands_typ : 	STRUCT
		xRaiseAlrComsDrive : BOOL;
		xRaiseAlrDriveError : BOOL;
		xRaiseAlrOvertorque : BOOL;
		xRaiseAlrDiffContact : BOOL;
		xRaiseControllerNotReady : BOOL;
	END_STRUCT;
	SimNonCrashParameters_typ : 	STRUCT
		iParameter : UINT;
	END_STRUCT;
	SimNonCrash_typ : 	STRUCT
		Commands : SimNonCrashCommands_typ;
		Parameters : SimNonCrashParameters_typ;
	END_STRUCT;
END_TYPE
```

### NonCrashSim.var - Local variables
```iecst
VAR
	iNonCrashSimIndex : USINT;
END_VAR
```

### TransVacuum.typ
```iecst
TYPE
	TransVacuumStatusCtrl :
		(
		TRANSVAC_OFF, (*Blower turned Off*)
		TRANSVAC_WAITING, (*The blower running at StartUp Duty cycle. IDLE state in previous programs*)
		TRANSVAC_CONTROLLING, (*Pressure beeing controlled by PID*)
		TRANSVAC_MAN,
		TRANSVAC_MAXIMUM (*Blowers working at 100% duty cycle*)
		);
	TransVacuumInputs_typ : 	STRUCT
		xPressureSensorError : BOOL;
		iPressureRaw : INT; (*Value from the input card*)
		xJointSystemPressure : BOOL; (*Digital vaccuum sensor signal . There is pressure enough in the system to close the joints*)
		xBlowersAnyCB : BOOL; (*Any Blower Circuit Breaker Nok*)
		xVaccAirFlow : BOOL; (*Flowmeter vacuum signal*)
		xSafetyEnable : BOOL; (*The Enable signals are active. Do not show alarms related to this if not active*)
	END_STRUCT;
	TransVacuumCommands_typ : 	STRUCT
		xRunProduction : BOOL; (*Signal to RUN in Auto Production mode. Signal to be keep while the running is wanted*)
		xRunJamRecovery : BOOL; (*Signal to RUN in Auto Jam Recovery mode. Signal to be keep while the running is wanted*)
		xRunByLine : BOOL; (*Signal to RUN in Auto mode. By LINE. Not production needed. Signal to be keep while the running is wanted*)
		xRunByRemote : BOOL; (*Signal to RUN in Auto mode. By REMOTE. Not production needed. Signal to be keep while the running is wanted*)
		xRunMaxDutyCycle : BOOL; (*Signal to RUN in Auto mode. Not production needed. Signal to be keep while the running is wanted. Set DutyCycle to 100%*)
		xMute : BOOL; (*command xMute *)
		xReset : BOOL; (*command xReset*)
	END_STRUCT;
	TransVacuumBlowerData_typ : 	STRUCT
		iIndex : USINT; (*Index of Inverters to control with this TransVacuum*)
		Direction : MotorDirection_enum; (*Direction of the motor to be run*)
	END_STRUCT;
	TransVacuumParamHw_typ : 	STRUCT
		uiNumBlowers : USINT := 1; (*Number of blowers in vacuum system*)
		xSystemWithJoints : BOOL; (*Define the system with joints and valves or without*)
		BlowerData : ARRAY[0..MAX_LAST_MOTOR_BLOWER]OF TransVacuumBlowerData_typ;
		iTotalAreas : USINT := 1; (*Total Number of areas in vacuum system*)
		rAreaWidth : REAL; (*The width of each area in mm*)
		rCentralAreaWithoutVacuum : REAL; (*Width of the central area with a pair of valves active, measured from the external tangent of the holes*)
	END_STRUCT;
	TransVacuumParameters_typ : 	STRUCT
		xInstalled : BOOL;
		rMaxSpeed : REAL; (*Maximum speed in the motor in rpm*)
		rMaxSystemVacuum : REAL; (*Maximum vacuum in mBar of the system to define the vacuum as Percentage*)
		Mode : StGeneral_States_Mode;
		AutoMode : stEFI_MachineAutoModes;
		parPID : stPIDParam;
		Hw : TransVacuumParamHw_typ;
		xExternalSafetyStop : BOOL; (*External Safety Stop order*)
		rStartUpDutyCycle : REAL := 60.0; (*Startup value of the Duty Cycle of the Blowers to Start if xStartUpEnable is active. GUI_I_ISTARTUPBLOWERDC*)
		xStartUpEnable : BOOL := FALSE; (*Start up state need in system*)
		xBeltRunning : BOOL; (*The belt in the machine is running. Used in Laboratory and ActiveOutOfProduction*)
		rMinDutyCycle : REAL;
		rMinVacPressureSetPointPerc : REAL; (*Maximum speed in the motor in rpm*)
		rVacPressureSetPointPerc : REAL := 50.0; (*SetPoint value of the desired pressure in the system in %. gui_i_iBlowerPressureSP*)
		rMaxPIDOut : REAL; (*Transvacuum pressure PID upper manipulated variable limit (upper modulation limit of the subsequent actuator)*)
		MinValvMask : UDINT; (*Minimum Vacuum valve mask open when working*)
	END_STRUCT;
	TransVacuumParametersSw_typ : 	STRUCT
		xActiveOutOfProduction : BOOL; (*Active the vacuum while in Automatic mode but not in Production*)
		rManSetPoint : REAL := 50.0; (*SetPoint value of working in manual. Value in %. Duty Cycle. gui_i_iManualBlowersPressureSP*)
		rVacPressureSetPointPerc : REAL := 50.0; (*SetPoint value of the desired pressure in the system in %. gui_i_iBlowerPressureSP*)
		ValvMask : UDINT; (*Vacuum valve mask from SW*)
	END_STRUCT;
	TransVacuumAlarms_typ : 	STRUCT
		xAlrVacuumSensor : BOOL; (*Error in the Vacuum sensor*)
		xAlrDriveBlowerError : BOOL; (*Error in the Drive managing the blower*)
		xWrnOvertorque : BOOL; (*Warning. Overtorque in the blower*)
		xAlrOvertorque : BOOL; (*Alarm. Overtorque in the blower*)
		xAlrComsBlower : BOOL; (*Not communication with the Drive of the blower*)
		xAlrJointSystemPressure : BOOL; (*Warning: Joint system underpressure*)
		xAlrBlowersAnyCB : BOOL; (*Warning: Blowers General Circuit Breaker*)
		xAlrBlowerCB : ARRAY[0..MAX_LAST_MOTOR_BLOWER]OF BOOL; (*Warning: Blowers Separate Circuit Breaker*)
		xAlrCommsBlower : ARRAY[0..MAX_LAST_MOTOR_BLOWER]OF BOOL; (*Alarm Comms Blower*)
		xAlrBlowerError : ARRAY[0..MAX_LAST_MOTOR_BLOWER]OF BOOL; (*Alarm Blower Error*)
		xAlrBlowerNotRunning : ARRAY[0..MAX_LAST_MOTOR_BLOWER]OF BOOL; (*Alarm Blower Not Running with Running order*)
	END_STRUCT;
	TransVacuumStatusBlower_typ : 	STRUCT
		rTorque : REAL := 1.0; (*Current torque N·m. gui_q_iCurrentTorque*)
		rDutyCycle : REAL; (*Current duty cycle %*)
		xMoving : BOOL; (*Started or Stopped*)
	END_STRUCT;
	TransVacuumStatus_typ : 	STRUCT
		State : TransVacuumStatusCtrl; (*State of the control*)
		Blower : TransVacuumStatusBlower_typ;
		Inverters : ARRAY[0..MAX_LAST_MOTOR_BLOWER]OF AxisP66_Status_typ;
		xInstalled : BOOL;
		rPressurePerc : REAL; (*Real pressure in %. Gui_q_iVacuumPressure*)
		rVacPressure : REAL; (*Real pressure in mbar*)
		xAtSpeed : BOOL;
		xStartedMan : BOOL;
		VacuumValves : UDINT; (*Active valves mask status*)
	END_STRUCT;
	TransVacuumOutputs_typ : 	STRUCT
		xActiveEvToEvacuateInk : BOOL; (*To active an Ev to evacuate the Ink inside the vacuum table*)
		VacuumValves : UDINT; (*2 integer var to control 20 valves; Least significative bits are in centring vacuum areas and most are in external areas.*)
	END_STRUCT;
	TransVacuum_typ : 	STRUCT
		Commands : TransVacuumCommands_typ;
		OrdersSw : TransVacuumOrdersSw_typ;
		Inputs : TransVacuumInputs_typ;
		Parameters : TransVacuumParameters_typ;
		parSw : TransVacuumParametersSw_typ;
		Status : TransVacuumStatus_typ;
		Alarms : TransVacuumAlarms_typ; (*Alarms*)
		AlSummary : stEFI_AlarmSummary; (*Alarms Summary*)
		Outputs : TransVacuumOutputs_typ;
	END_STRUCT;
	TransVacuumOrdersSw_typ : 	STRUCT
		xRunManual : BOOL; (*Signal to RUN in Manual mode. Signal to be keep while the running is wanted*)
	END_STRUCT;
END_TYPE
```

### TransVacuum.var
```iecst
VAR
	iIndexTransVacuum : USINT;
END_VAR
```

### Program Logical/ExtPack/_Transport/TransVacuumCtrl/TransVacuumCtrl_v1/InitTransVacuumCtrl (IEC)

#### InitTransVacuumCtrl.st - Cyclic code
```iecst
PROGRAM _CYCLIC
	//Init the index to work with
	 iIndexTransVacuum := 1;
END_PROGRAM
```

### Program Logical/ExtPack/_Transport/TransVacuumCtrl/TransVacuumCtrl_v1/TransVacuumCtrl (IEC)

#### TransVacuumCtrl.st - Init, cyclic, exit code
```iecst
PROGRAM _CYCLIC

	//References of the program
	dataVacc ACCESS ADR (gTransVacuum[iIndexTransVacuum]);

	dataVacc.Status.xInstalled := dataVacc.Parameters.xInstalled;

	//Check if there is any blower enabled. If all blowers disabled, consider it as not installed
	xAllBlowerDisabled := TRUE;
	FOR uiIndex := 1 TO dataVacc.Parameters.Hw.uiNumBlowers BY 1 DO
		IF NOT xDisableBlower[uiIndex] THEN
			xAllBlowerDisabled := FALSE;
		END_IF
	END_FOR

	IF NOT dataVacc.Status.xInstalled OR xAllBlowerDisabled THEN
		ResetAlarms;
		ResetCommands;
		iIndexTransVacuum:= iIndexTransVacuum +1;
		RETURN;
	END_IF

	//Reset alarms
	IF dataVacc.Commands.xReset THEN
		ResetAlarms;
	END_IF

	// Variables Summary
	xProductionOrJamRecovery := dataVacc.Parameters.AutoMode.xProduction OR dataVacc.Parameters.AutoMode.xJamRecovery;

	//Limit of the configured blowers used. It must be inside the array size
	dataVacc.Parameters.Hw.uiNumBlowers := LIMIT(1, dataVacc.Parameters.Hw.uiNumBlowers, MAX_LAST_MOTOR_BLOWER);
	dataVacc.Parameters.rMaxPIDOut := LIMIT(30, dataVacc.Parameters.rMaxPIDOut, 100); // Limit to 30 to avoid the blowers not starting

	// INPUTS
	//PRESURE SENSOR FILTER LOW PASS
	FLP_PresFilterPasLow.CutOffFrequency := 0.2;
	FLP_PresFilterPasLow.Order := 3;
	FLP_PresFilterPasLow.Type := mtFILTER_BESSEL;
	FLP_PresFilterPasLow.Enable := TRUE;

	FLP_PresFilterPasLow.In := INT_TO_REAL(dataVacc.Inputs.iPressureRaw);
	FLP_PresFilterPasLow();
	FLP_PresFilterPasLow.Update := FALSE;

	rVacPressure := -1*(FLP_PresFilterPasLow.Out -16384.0)/16384.0*150.0;

	rVacPressurePerc := 100 * ABS(rVacPressure/dataVacc.Parameters.rMaxSystemVacuum);

	StateManager;

	PressureCtrl;

	//////////////////////////////////////////////////////////////////
	// BLOWERS BLOWERS BLOWERS BLOWERS BLOWERS BLOWERS BLOWERS BLOWERS
	/////////////////////////////////////////////////////////////////
	xAllBlowersRunning := TRUE;
	xAllBlowersAtSpeed := TRUE;
	FOR uiIndex := 1 TO dataVacc.Parameters.Hw.uiNumBlowers BY 1 DO
		//Reference to the motor of the blower
		Blower ACCESS ADR(gAxisInverter[dataVacc.Parameters.Hw.BlowerData[uiIndex].iIndex]);
		BlowerDirection := dataVacc.Parameters.Hw.BlowerData[uiIndex].Direction;
		ConditionStart_copy := ConditionsStart_copy[uiIndex];

		//Show data in Status
		dataVacc.Status.Inverters[uiIndex] := Blower.Status;

		//Copy working element to watch it
		BlowersWatch[uiIndex] := Blower;
		BlowerDirectionsWatch[uiIndex] := BlowerDirection;

		//Give the option to disable one of the blowers if it is damaged
		IF NOT xDisableBlower[uiIndex] THEN
			BlowerAlarms;
			BlowerControl;
		END_IF

		//Store the values from Blower Control to use edges
		ConditionsStart_copy[uiIndex] := ConditionStart;
	END_FOR

	//Delaying the signal to be sure we have vaccuum in the system when activating the signal
	tonBlowersRunning.IN := xAllBlowersRunning;
	tonBlowersRunning.PT := t#2s;
	tonBlowersRunning();
	dataVacc.Status.Blower.xMoving := tonBlowersRunning.Q;

	Alarms;

	//Define the status of the Structure
	dataVacc.Status.State	:= StatusCtrl;
	dataVacc.Status.rVacPressure := rVacPressure;
	dataVacc.Status.rPressurePerc := 100 * ABS(rVacPressure/dataVacc.Parameters.rMaxSystemVacuum);
	dataVacc.Status.xAtSpeed := xAllBlowersAtSpeed;

	//Evacuate ink inside vacuum's table
	tpEvEvacuateInk.IN := EDGEPOS(StatusCtrl=TRANSVAC_OFF);
	tpEvEvacuateInk.PT := T#1h;
	tpEvEvacuateInk();
	dataVacc.Outputs.xActiveEvToEvacuateInk := StatusCtrl=TRANSVAC_OFF; // AND tpEvEvacuateInk.Q; //Mechanical team wants this ev active as long as vacuum is stopped

	dataVacc.Commands.xReset := FALSE;
	StatusCtrl_copy := StatusCtrl;

	iIndexTransVacuum := iIndexTransVacuum + 1;

END_PROGRAM
```

#### StateManager.st
```iecst
ACTION StateManager:

//	TRANSVAC_OFF				Blower turned Off
//	TRANSVAC_WAITING			The blower running at StartUp Duty cycle. IDLE state in previous programs
//	TRANSVAC_CONTROLLING		Pressure beeing controlled BY PID
//	TRANSVAC_MAN

	// Order not in production
	iReasonOutOfProduction.0 := dataVacc.parSw.xActiveOutOfProduction AND dataVacc.Parameters.AutoMode.xBypass;

	//Memorice first start in laboratory mode. This line is needed before the memory is uesd
	IF xRunBlowerAuto THEN xLabStartedBlowers := dataVacc.Parameters.AutoMode.xLaboratory; ELSE xLabStartedBlowers := FALSE; END_IF
	iReasonOutOfProduction.1 := dataVacc.parSw.xActiveOutOfProduction AND dataVacc.Parameters.AutoMode.xLaboratory AND
								(dataVacc.Parameters.xBeltRunning OR xLabStartedBlowers);

	iReasonOutOfProduction.2 := dataVacc.Commands.xRunByLine;
	iReasonOutOfProduction.3 := dataVacc.Commands.xRunByRemote;

	xRunOutOfProduction := iReasonOutOfProduction > 0;

	////////////////Auto Order
	iReasonRunAuto.0 := dataVacc.Commands.xRunProduction AND dataVacc.Parameters.AutoMode.xProduction;
	iReasonRunAuto.1 := dataVacc.Parameters.Mode.xAuto AND xRunOutOfProduction;
	iReasonRunAuto.2 := dataVacc.Commands.xRunJamRecovery AND dataVacc.Parameters.AutoMode.xJamRecovery;
	xRunBlowerAuto := iReasonRunAuto > 0;

	////////////////Manual order
	xRunBlowerMan := dataVacc.Parameters.Mode.xManual AND dataVacc.OrdersSw.xRunManual; //To avoid blowers starts again after restoring STOs if blowers were running when STOs were switched off

	CASE StatusCtrl OF

		TRANSVAC_OFF:
			IF NOT tofNotStartAfterEStop.Q THEN
				IF EDGEPOS(xRunBlowerMan) THEN
					StatusCtrl:=TRANSVAC_MAN;
				END_IF

				IF xRunBlowerAuto AND (dataVacc.parSw.rVacPressureSetPointPerc>=dataVacc.Parameters.rMinVacPressureSetPointPerc) THEN
					IF dataVacc.Parameters.xStartUpEnable THEN
						StatusCtrl:=TRANSVAC_WAITING;
					ELSE
						StatusCtrl:=TRANSVAC_CONTROLLING;
					END_IF
				END_IF
			END_IF

		TRANSVAC_WAITING:
			IF rVacPressurePerc > dataVacc.Parameters.rVacPressureSetPointPerc THEN
				StatusCtrl:=TRANSVAC_CONTROLLING;
			END_IF
			IF dataVacc.Commands.xRunMaxDutyCycle THEN
				StatusCtrl:=TRANSVAC_MAXIMUM;
			END_IF

			GoToOffIfNotAutoOrSP;

		TRANSVAC_CONTROLLING:
			IF dataVacc.Parameters.xStartUpEnable AND (dataVacc.Status.Blower.rDutyCycle > dataVacc.Parameters.rStartUpDutyCycle) THEN
				StatusCtrl:=TRANSVAC_WAITING;
			END_IF
			IF dataVacc.Commands.xRunMaxDutyCycle THEN
				StatusCtrl:=TRANSVAC_MAXIMUM;
			END_IF

			GoToOffIfNotAutoOrSP;

		TRANSVAC_MAXIMUM:
			IF xRunBlowerAuto THEN
				StatusCtrl:=TRANSVAC_CONTROLLING;
			ELSIF NOT dataVacc.Commands.xRunMaxDutyCycle AND NOT xRunBlowerAuto THEN
				StatusCtrl:=TRANSVAC_OFF;
			END_IF

		TRANSVAC_MAN:
			IF NOT xRunBlowerMan THEN
				StatusCtrl:=TRANSVAC_OFF;
				dataVacc.Status.xStartedMan := FALSE;
			END_IF

	END_CASE

	//In Zero, always stop blowers
	IF dataVacc.Parameters.Mode.xZero OR dataVacc.Parameters.xExternalSafetyStop THEN
		StatusCtrl:=TRANSVAC_OFF;
		ResetCommands;
	END_IF

	// Timer to be sure not start the blowers after 6 seconds after recovering from a Safety Signal
	tofNotStartAfterEStop.IN := EDGENEG(dataVacc.Parameters.xExternalSafetyStop);
	tofNotStartAfterEStop.PT := T#0s;
	tofNotStartAfterEStop();

	//Just with the status of manual
	dataVacc.Status.xStartedMan := StatusCtrl = TRANSVAC_MAN;

END_ACTION

ACTION GoToOffIfNotAutoOrSP:

	TON_StopBlowersDly.IN:= NOT xRunBlowerAuto OR (dataVacc.Parameters.rMinVacPressureSetPointPerc > dataVacc.parSw.rVacPressureSetPointPerc);
	TON_StopBlowersDly.PT:= t#200ms;
	TON_StopBlowersDly();

	IF TON_StopBlowersDly.Q THEN
		StatusCtrl:=TRANSVAC_OFF;
	END_IF

END_ACTION

ACTION ResetCommands:
	IF NOT dataVacc.Commands.xReset THEN
		dataVacc.Commands := CommandsReseted;
	ELSE
		dataVacc.Commands := CommandsReseted;
		dataVacc.Commands.xReset := TRUE;
	END_IF
END_ACTION
```
